DATA_BLOCK "ErrTextList"   // DB371
{ S7_Optimized_Access := 'TRUE' }
// stored: AutoNumber false, MemoryReserve 0
   VAR RETAIN
      language : Array[1..10] of WString[2];   // language for alarm text [ISO639-1]
   END_VAR
   VAR
      writeMessage : Bool;   // write message from program to data block
      err : Array[2000..2205] of Struct   // alarm text
         idProd : UInt;   // producer Id (for Plc: 0=Program_Alarm, 4=SysDiag, 5=MotionControl, 6=Security, 8=GRAPH, 9=ProDiag)
         id : UInt;   // alarm Id
         prio : UInt;   // 0 .. 16 (0-1=info, 2=safety, 3=warning, 4-16=fault)
         alarm : Array[1..8] of WString[150];   // alarm text
      END_STRUCT;
   END_VAR
BEGIN
   language[1] := WSTRING#'de';
   language[2] := WSTRING#'en';
   language[3] := WSTRING#'it';
   language[4] := WSTRING#'fr';
   language[5] := WSTRING#'es';
   err[2031..2040].idProd := 0;
   err[2160..2167].idProd := 0;
   err[2170..2177].idProd := 0;
   err[2180..2187].idProd := 0;
   err[2031..2040].id := 0;
   err[2160..2167].id := 0;
   err[2170..2177].id := 0;
   err[2180..2187].id := 0;
   err[2000..2002].prio := 2;
   err[2004..2005].prio := 2;
   err[2010..2011].prio := 2;
   err[2013..2014].prio := 2;
   err[2016..2017].prio := 2;
   err[2019..2020].prio := 2;
   err[2030..2031].prio := 2;
   err[2032].prio := 0;
   err[2033..2040].prio := 2;
   err[2050].prio := 1;
   err[2052].prio := 0;
   err[2054].prio := 1;
   err[2060].prio := 10;
   err[2075].prio := 2;
   err[2080..2083].prio := 11;
   err[2090..2091].prio := 9;
   err[2100..2102].prio := 10;
   err[2110].prio := 8;
   err[2111].prio := 0;
   err[2120].prio := 12;
   err[2121..2125].prio := 7;
   err[2150].prio := 11;
   err[2151].prio := 10;
   err[2152..2153].prio := 8;
   err[2154].prio := 1;
   err[2156].prio := 1;
   err[2160].prio := 11;
   err[2161].prio := 10;
   err[2162..2163].prio := 8;
   err[2164].prio := 1;
   err[2165].prio := 0;
   err[2166].prio := 1;
   err[2167].prio := 0;
   err[2170].prio := 11;
   err[2171].prio := 10;
   err[2172..2173].prio := 8;
   err[2174].prio := 1;
   err[2175].prio := 0;
   err[2176].prio := 1;
   err[2177].prio := 0;
   err[2180].prio := 11;
   err[2181].prio := 10;
   err[2182..2183].prio := 8;
   err[2184].prio := 1;
   err[2185].prio := 0;
   err[2186].prio := 1;
   err[2187].prio := 0;
   err[2189].prio := 8;
   err[2190].prio := 9;
   err[2000].alarm[1] := WSTRING#'PLC - Not Aus Taster gedrückt am Pc Terminal (-14SB0+HMI.GLD)';
   err[2000].alarm[2] := WSTRING#'PLC - Emergency stop pressed at Pc terminal (-14SB0+HMI.GLD)';
   err[2000].alarm[3] := WSTRING#'PLC - Tasto per arresto di emergenza premuto sul terminale Pc (-14SB0+HMI.GLD)';
   err[2000].alarm[4] := WSTRING#'PLC - Arrêt d`urgence appuyé sur le terminal PC (-14SB0+HMI.GLD)';
   err[2000].alarm[5] := WSTRING#'PLC - Parada de emergencia presionada en terminal Pc (-14SB0+HMI.GLD)';
   err[2001].alarm[1] := WSTRING#'PLC - Not Aus Schlüsselschalter ausgeschalten am Pc Terminal (-14SB1+HMI.GLD)';
   err[2001].alarm[2] := WSTRING#'PLC - Emergency enable key switch off at Pc terminal (-14SB1+HMI.GLD)';
   err[2001].alarm[3] := WSTRING#'PLC - Interruttore a chiave per aresto di emergenza spento sul terminale del PC (-14SB1+HMI.GLD)';
   err[2001].alarm[4] := WSTRING#'PLC - Interrupteur d`urgence désactivé sur le terminal PC (-14SB1+HMI.GLD)';
   err[2001].alarm[5] := WSTRING#'PLC - Interruptor de llave de parada de emergencia apagado en la terminal de la PC (-14SB1+HMI.GLD)';
   err[2002].alarm[1] := WSTRING#'PLC - Quittierung notwendig für Not Aus Taster/Schlüsselschalter am Pc Terminal (-14SB0/1+HMI.GLD)';
   err[2002].alarm[2] := WSTRING#'PLC - Acknowledge required for emergency stop/key switch at Pc terminal (-14SB0/1+HMI.GLD)';
   err[2002].alarm[3] := WSTRING#'PLC - Reset richiesto per pulsante/interrutore di arresto di emergenza sul terminale PC (-14SB0/1+HMI.GLD)';
   err[2002].alarm[4] := WSTRING#'PLC - Reconnaissance nécessaire pour l`arrêt d`urgence/interrupteur à clé sur le terminal PC (-14SB0/1+HMI.GLD)';
   err[2002].alarm[5] := WSTRING#'PLC - Es necesario reiniciar para el botónIinterruptor de emergencia en terminal de PC (-14SB0/1+HMI.GLD)';
   err[2004].alarm[1] := WSTRING#'PLC - Not Aus von externe machine (-XNA+SGV) - aktiv';
   err[2004].alarm[2] := WSTRING#'PLC - Emergency stop from external machine (-XNA+SGV) - active';
   err[2004].alarm[3] := WSTRING#'PLC - Arresto di emergenza da macchina esterna (-XNA+SGV) - attivo';
   err[2004].alarm[4] := WSTRING#'PLC - Arrêt d`urgence depuis une machine externe (-XNA+SGV) - actif';
   err[2004].alarm[5] := WSTRING#'PLC - Parada de emergencia desde máquina externa (-XNA+SGV) - activo';
   err[2005].alarm[1] := WSTRING#'PLC - Not Aus von externe machine (-XNA+SGV) - Quittierung notwendig';
   err[2005].alarm[2] := WSTRING#'PLC - Emergency stop from external machine (-XNA+SGV) - acknowledgement required';
   err[2005].alarm[3] := WSTRING#'PLC - Arresto di emergenza da macchina esterna (-XNA+SGV) - reset necessario';
   err[2005].alarm[4] := WSTRING#'PLC - Arrêt d`urgence depuis une machine externe (-XNA+SGV) - réinitialiser requis';
   err[2005].alarm[5] := WSTRING#'PLC - Parada de emergencia desde máquina externa (-XNA+SGV) - es necesario reiniciar';
   err[2010].alarm[1] := WSTRING#'PLC - Sicherheitsschalter -14SS1.TL+SGV bei Scanner für visuelle Beurteilung oben links - open';
   err[2010].alarm[2] := WSTRING#'PLC - Safety switch -14SS1.TL+SGV at scanner for visual measurement top left - open';
   err[2010].alarm[3] := WSTRING#'PLC - Interruttore di sicurezza -14SS1.TL+SGV sullo scanner per misurazione visiva in alto a sinistra - aperto';
   err[2010].alarm[4] := WSTRING#'PLC - interrupteur de sécurité -14SS1.TL+SGV au scanner pour mesure visuelle en haut à gauche - ouvert';
   err[2010].alarm[5] := WSTRING#'PLC - interruptor de seguridad -14SS1.TL+SGV en el escáner para medición visual arriba a la izquierda - abierto';
   err[2011].alarm[1] := WSTRING#'PLC - Sicherheitsschalter -14SS1.TL+SGV bei Scanner für visuelle Beurteilung oben links - Quittierung notwendig';
   err[2011].alarm[2] := WSTRING#'PLC - safety switch -14SS1.TL+SGV at scanner for visual measurement top left - acknowledge required';
   err[2011].alarm[3] := WSTRING#'PLC - Interruttore di sicurezza -14SS1.TL+SGV sullo scanner per misurazione visiva in alto a sinistra - reset necessario';
   err[2011].alarm[4] := WSTRING#'PLC - interrupteur de sécurité -14SS1.TL+SGV au scanner pour mesure visuelle en haut à gauche - réinitialiser requis';
   err[2011].alarm[5] := WSTRING#'PLC - interruptor de seguridad -14SS1.TL+SGV en el escáner para medición visual arriba a la izquierda - es necesario reiniciar';
   err[2013].alarm[1] := WSTRING#'PLC - Sicherheitsschalter -14SS1.BL+SGV bei Scanner für visuelle Beurteilung unten links - open';
   err[2013].alarm[2] := WSTRING#'PLC - Safety switch -14SS1.BL+SGV at scanner for visual measurement bottom left - open';
   err[2013].alarm[3] := WSTRING#'PLC - Interruttore di sicurezza -14SS1.BL+SGV sullo scanner per misurazione visiva in basso a sinistra - aperto';
   err[2013].alarm[4] := WSTRING#'PLC - interrupteur de sécurité -14SS1.BL+SGV au scanner pour mesure visuelle en bas à gauche - ouvert';
   err[2013].alarm[5] := WSTRING#'PLC - interruptor de seguridad -14SS1.BL+SGV en el escáner para medición visual abajoa la izquierda - abierto';
   err[2014].alarm[1] := WSTRING#'PLC - Sicherheitsschalter -14SS1.BL+SGV bei Scanner für visuelle Beurteilung unten links - Quittierung notwendig';
   err[2014].alarm[2] := WSTRING#'PLC - Safety switch -14SS1.BL+SGV at scanner for visual measurement bottom left - acknowledge required';
   err[2014].alarm[3] := WSTRING#'PLC - Interruttore di sicurezza -14SS1.BL+SGV sullo scanner per misurazione visiva in basso a sinistra - reset necessario';
   err[2014].alarm[4] := WSTRING#'PLC - interrupteur de sécurité -14SS1.BL+SGV au scanner pour mesure visuelle en bas à gauche - réinitialiser requis';
   err[2014].alarm[5] := WSTRING#'PLC - interruptor de seguridad -14SS1.BL+SGV en el escáner para medición visual abajoa la izquierda - es necesario reiniciar';
   err[2016].alarm[1] := WSTRING#'PLC - Sicherheitsschalter -14SS1.TR+SGV bei Scanner für visuelle Beurteilung oben rechts- open';
   err[2016].alarm[2] := WSTRING#'PLC - Safety switch -14SS1.TR+SGV at scanner for visual measurement top right - open';
   err[2016].alarm[3] := WSTRING#'PLC - Interruttore di sicurezza -14SS1.TR+SGV sullo scanner per misurazione visiva in alto a destra - aperto';
   err[2016].alarm[4] := WSTRING#'PLC - interrupteur de sécurité -14SS1.TR+SGV au scanner pour mesure visuelle en haut à droite - ouvert';
   err[2016].alarm[5] := WSTRING#'PLC - interruptor de seguridad -14SS1.TR+SGV en el escáner para medición visual arriba a la derecha - abierto';
   err[2017].alarm[1] := WSTRING#'PLC - Sicherheitsschalter -14SS1.TR+SGV bei Scanner für visuelle Beurteilung oben rechts- Quittierung notwendig';
   err[2017].alarm[2] := WSTRING#'PLC - Safety switch -14SS1.TR+SGV at scanner for visual measurement top right -  acknowledge required';
   err[2017].alarm[3] := WSTRING#'PLC - Interruttore di sicurezza -14SS1.TR+SGV sullo scanner per misurazione visiva in alto a destra - reset necessario';
   err[2017].alarm[4] := WSTRING#'PLC - interrupteur de sécurité -14SS1.TR+SGV au scanner pour mesure visuelle en haut à droite - réinitialiser requis';
   err[2017].alarm[5] := WSTRING#'PLC - interruptor de seguridad -14SS1.TR+SGV en el escáner para medición visual arriba a la derecha - es necesario reiniciar';
   err[2019].alarm[1] := WSTRING#'PLC - Sicherheitsschalter -14SS1.BR+SGV bei Scanner für visuelle Beurteilung unten rechts - open';
   err[2019].alarm[2] := WSTRING#'PLC - Safety switch -14SS1.BR+SGV at scanner for visual measurement bottom right - open';
   err[2019].alarm[3] := WSTRING#'PLC - Interruttore di sicurezza -14SS1.BR+SGV sullo scanner per misurazione visiva in basso a destra - aperto';
   err[2019].alarm[4] := WSTRING#'PLC - interrupteur de sécurité -14SS1.BR+SGV au scanner pour mesure visuelle en bas à droite - ouvert';
   err[2019].alarm[5] := WSTRING#'PLC - interruptor de seguridad -14SS1.BR+SGV en el escáner para medición visual abajo a la derecha - abierto';
   err[2020].alarm[1] := WSTRING#'PLC - Sicherheitsschalter -14SS1.BR+SGV bei Scanner für visuelle Beurteilung unten rechts - Quittierung notwendig';
   err[2020].alarm[2] := WSTRING#'PLC - Safety switch -14SS1.BR+SGV at scanner for visual measurement bottom right -  acknowledge required';
   err[2020].alarm[3] := WSTRING#'PLC - Interruttore di sicurezza -14SS1.BR+SGV sullo scanner per misurazione visiva in basso a destra - reset necessario';
   err[2020].alarm[4] := WSTRING#'PLC - interrupteur de sécurité -14SS1.BR+SGV au scanner pour mesure visuelle en bas à droite - réinitialiser requis';
   err[2020].alarm[5] := WSTRING#'PLC - interruptor de seguridad -14SS1.BR+SGV en el escáner para medición visual abajo a la derecha - es necesario reiniciar';
   err[2030].alarm[1] := WSTRING#'PLC - Sicherheitsschalter -14SS1.TL+SGX bei Scanner für X-Ray oben links - open';
   err[2030].alarm[2] := WSTRING#'PLC - Safety switch -14SS1.TL+SGX at scanner for X-Ray top left - open';
   err[2030].alarm[3] := WSTRING#'PLC - Interruttore di sicurezza -14SS1.TL+SGX sullo scanner per X-Ray in alto a sinistra - aperto';
   err[2030].alarm[4] := WSTRING#'PLC - interrupteur de sécurité -14SS1.TL+SGX au scanner pour X-Ray en haut à gauche - ouvert';
   err[2030].alarm[5] := WSTRING#'PLC - interruptor de seguridad -14SS1.TL+SGX en el escáner para X-Ray arriba a la izquierda - abierto';
   err[2030].alarm[6..8] := WSTRING#'';
   err[2031].alarm[1] := WSTRING#'PLC - Sicherheitsschalter -14SS1.TL+SGX bei Scanner für X-Ray oben links - Quittierung notwendig';
   err[2031].alarm[2] := WSTRING#'PLC - safety switch -14SS1.TL+SGX at scanner for X-Ray top left - acknowledge required';
   err[2031].alarm[3] := WSTRING#'PLC - Interruttore di sicurezza -14SS1.TL+SGX sullo scanner per X-Ray in alto a sinistra - reset necessario';
   err[2031].alarm[4] := WSTRING#'PLC - interrupteur de sécurité -14SS1.TL+SGX au scanner pour X-Ray en haut à gauche - réinitialiser requis';
   err[2031].alarm[5] := WSTRING#'PLC - interruptor de seguridad -14SS1.TL+SGX en el escáner para X-Ray arriba a la izquierda - es necesario reiniciar';
   err[2031].alarm[6..8] := WSTRING#'';
   err[2032].alarm[1..8] := WSTRING#'';
   err[2033].alarm[1] := WSTRING#'PLC - Sicherheitsschalter -14SS1.BL+SGX bei Scanner für X-Ray unten links - open';
   err[2033].alarm[2] := WSTRING#'PLC - Safety switch -14SS1.BL+SGX at scanner for X-Ray bottom left - open';
   err[2033].alarm[3] := WSTRING#'PLC - Interruttore di sicurezza -14SS1.BL+SGX sullo scanner per X-Ray in basso a sinistra - aperto';
   err[2033].alarm[4] := WSTRING#'PLC - interrupteur de sécurité -14SS1.BL+SGX au scanner pour X-Ray en bas à gauche - ouvert';
   err[2033].alarm[5] := WSTRING#'PLC - interruptor de seguridad -14SS1.BL+SGX en el escáner para X-Ray abajoa la izquierda - abierto';
   err[2033].alarm[6..8] := WSTRING#'';
   err[2034].alarm[1] := WSTRING#'PLC - Sicherheitsschalter -14SS1.BL+SGX bei Scanner für X-Ray unten links - Quittierung notwendig';
   err[2034].alarm[2] := WSTRING#'PLC - Safety switch -14SS1.BL+SGX at scanner for X-Rayt bottom left - acknowledge required';
   err[2034].alarm[3] := WSTRING#'PLC - Interruttore di sicurezza -14SS1.BL+SGX sullo scanner per X-Ray in basso a sinistra - reset necessario';
   err[2034].alarm[4] := WSTRING#'PLC - interrupteur de sécurité -14SS1.BL+SGX au scanner pour X-Ray en bas à gauche - réinitialiser requis';
   err[2034].alarm[5] := WSTRING#'PLC - interruptor de seguridad -14SS1.BL+SGX en el escáner para X-Ray abajoa la izquierda - es necesario reiniciar';
   err[2034].alarm[6..8] := WSTRING#'';
   err[2035].alarm[1..8] := WSTRING#'';
   err[2036].alarm[1] := WSTRING#'PLC - Sicherheitsschalter -14SS1.TR+SGX bei Scanner für X-Ray oben rechts- open';
   err[2036].alarm[2] := WSTRING#'PLC - Safety switch -14SS1.TR+SGX at scanner for X-Ray top right - open';
   err[2036].alarm[3] := WSTRING#'PLC - Interruttore di sicurezza -14SS1.TR+SGX sullo scanner per X-Ray in alto a destra - aperto';
   err[2036].alarm[4] := WSTRING#'PLC - interrupteur de sécurité -14SS1.TR+SGX au scanner pour X-Ray en haut à droite - ouvert';
   err[2036].alarm[5] := WSTRING#'PLC - interruptor de seguridad -14SS1.TR+SGX en el escáner para X-Ray arriba a la derecha - abierto';
   err[2036].alarm[6..8] := WSTRING#'';
   err[2037].alarm[1] := WSTRING#'PLC - Sicherheitsschalter -14SS1.TR+SGX bei Scanner für X-Ray oben rechts- Quittierung notwendig';
   err[2037].alarm[2] := WSTRING#'PLC - Safety switch -14SS1.TR+SGX at scanner for X-Ray top right -  acknowledge required';
   err[2037].alarm[3] := WSTRING#'PLC - Interruttore di sicurezza -14SS1.TR+SGX sullo scanner per X-Ray in alto a destra - reset necessario';
   err[2037].alarm[4] := WSTRING#'PLC - interrupteur de sécurité -14SS1.TR+SGX au scanner pour X-Ray en haut à droite - réinitialiser requis';
   err[2037].alarm[5] := WSTRING#'PLC - interruptor de seguridad -14SS1.TR+SGX en el escáner para X-Ray arriba a la derecha - es necesario reiniciar';
   err[2037].alarm[6..8] := WSTRING#'';
   err[2038].alarm[1..8] := WSTRING#'';
   err[2039].alarm[1] := WSTRING#'PLC - Sicherheitsschalter -14SS1.BR+SGX bei Scanner für X-Ray unten rechts - open';
   err[2039].alarm[2] := WSTRING#'PLC - Safety switch -14SS1.BR+SGX at scanner for X-Ray bottom right - open';
   err[2039].alarm[3] := WSTRING#'PLC - Interruttore di sicurezza -14SS1.BR+SGX sullo scanner per X-Ray in basso a destra - aperto';
   err[2039].alarm[4] := WSTRING#'PLC - interrupteur de sécurité -14SS1.BR+SGX au scanner pour X-Ray en bas à droite - ouvert';
   err[2039].alarm[5] := WSTRING#'PLC - interruptor de seguridad -14SS1.BR+SGX en el escáner para X-Ray abajo a la derecha - abierto';
   err[2039].alarm[6..8] := WSTRING#'';
   err[2040].alarm[1] := WSTRING#'PLC - Sicherheitsschalter -14SS1.BR+SGX bei Scanner für X-Ray unten rechts - Quittierung notwendig';
   err[2040].alarm[2] := WSTRING#'PLC - Safety switch -14SS1.BR+SGX at scanner for X-Ray bottom right -  acknowledge required';
   err[2040].alarm[3] := WSTRING#'PLC - Interruttore di sicurezza -14SS1.BR+SGX sullo scanner per X-Ray in basso a destra - reset necessario';
   err[2040].alarm[4] := WSTRING#'PLC - interrupteur de sécurité -14SS1.BR+SGX au scanner pour X-Ray en bas à droite - réinitialiser requis';
   err[2040].alarm[5] := WSTRING#'PLC - interruptor de seguridad -14SS1.BR+SGX en el escáner para X-Ray abajo a la derecha - es necesario reiniciar';
   err[2050].alarm[1] := WSTRING#'PLC - Schlüsselschalter für Einrichtbetrieb am Scanner links aktiviert (-14SB1+SSTL)';
   err[2050].alarm[2] := WSTRING#'PLC - setting mode key switch at scanner left active (-14SB1+SSTL)';
   err[2050].alarm[3] := WSTRING#'PLC - Interruttore a chiave per la modalità di impostazione attivato sullo scanner a sinistra (-14SB1+SSTL)';
   err[2050].alarm[4] := WSTRING#'PLC - commutateur à clé du mode de réglage à gauche du scanner actif (-14SB1+SSTL)';
   err[2050].alarm[5] := WSTRING#'PLC - interruptor de modo de ajuste a la izquierda del escáner activo (-14SB1+SSTL)';
   err[2052].alarm[1] := WSTRING#'PLC - Taster für Freigabe Verstellungen am Scanner links aktiviert (-14SB2+SSTL)';
   err[2052].alarm[2] := WSTRING#'PLC - button to enable adjustments at scanner left active (-14SB21+SSTL)';
   err[2052].alarm[3] := WSTRING#'PLC - pulsante per abilitare le assi attivato sullo scanner a sinistra (-14SB2+SSTL)';
   err[2052].alarm[4] := WSTRING#'PLC - bouton pour activer les réglages à gauche du scanner actif (-14SB2+SSTL)';
   err[2052].alarm[5] := WSTRING#'PLC - botón para habilitar ajustes a la izquierda del escáner activo (-14SB2+SSTL)';
   err[2054].alarm[1] := WSTRING#'PLC - Kühlgeräte wurden am Scanner rechts deaktiviert (-14SB2+SSTL)';
   err[2054].alarm[2] := WSTRING#'PLC - air-conditioning is switched off at scanner right (-0SH1+SSTR)';
   err[2054].alarm[3] := WSTRING#'PLC - l`aria condizionata è stata spenta sullo scanner a destra (-14SB2+SSTL)';
   err[2054].alarm[4] := WSTRING#'PLC - la climatisation est éteinte au niveau du scanner à droite (-14SB2+SSTL)';
   err[2054].alarm[5] := WSTRING#'PLC - El aire acondicionado está apagado en el escáner a la derecha (-14SB2+SSTL)';
   err[2060].alarm[1] := WSTRING#'PLC - Störung Sicherheitsmodule';
   err[2060].alarm[2] := WSTRING#'PLC - fault safety modules plc';
   err[2060].alarm[3] := WSTRING#'PLC - errore sui moduli di sicurezza';
   err[2060].alarm[4] := WSTRING#'PLC - modules de sécurité contre les défauts';
   err[2060].alarm[5] := WSTRING#'PLC - módulos de seguridad contra fallas';
   err[2075].alarm[1] := WSTRING#'PLC - Sicherheitsbereich Extern oder Intern ausgeschalten - Quittierung notwendig';
   err[2075].alarm[2] := WSTRING#'PLC - safety area internal/external switched off - acknowledge required';
   err[2075].alarm[3] := WSTRING#'PLC - area di sicurezza interna/esterna spenta- reset necessario';
   err[2075].alarm[4] := WSTRING#'PLC - zone de sécurité interne/externe désactivée - réinitialiser requis';
   err[2075].alarm[5] := WSTRING#'PLC - area de seguridad interna/externa apagada - es necesario reiniciar';
   err[2080].alarm[1] := WSTRING#'PLC - Störung Rückführung Sicherheitsbereich - Bereich laser (-14KA1+SGV)';
   err[2080].alarm[2] := WSTRING#'PLC - fault safety feedback monitoring - area laser (-14KA1+SGV)';
   err[2080].alarm[3] := WSTRING#'PLC - errore monitoraggio feedback di sicurezza - area laser (-14KA1+SGV)';
   err[2080].alarm[4] := WSTRING#'PLC - défaut surveillance de la sécurité - zone laser (-14KA1+SGV)';
   err[2080].alarm[5] := WSTRING#'PLC - fallo de monitoreo de retroalimentación de seguridad - área de láser (-14KA1+SGV)';
   err[2081].alarm[1] := WSTRING#'PLC - Störung Rückführung Sicherheitsbereich - Bereich Verstellung (-14KA2+SGV)';
   err[2081].alarm[2] := WSTRING#'PLC - fault safety feedback monitoring - area adjustment (-14KA2+SGV)';
   err[2081].alarm[3] := WSTRING#'PLC - errore monitoraggio feedback di sicurezza - area posizionamento (-14KA2+SGV)';
   err[2081].alarm[4] := WSTRING#'PLC - défaut surveillance de la sécurité - zone réglage (-14KA2+SGV)';
   err[2081].alarm[5] := WSTRING#'PLC - fallo de monitoreo de retroalimentación de seguridad - área de ajuste (-14KA2+SGV)';
   err[2082].alarm[1] := WSTRING#'PLC - Störung Rückführung Sicherheitsbereich - Bereich Verstellung LINMOT (8U1+SGV)';
   err[2082].alarm[2] := WSTRING#'PLC - fault safety feedback monitoring - area adjustment LINMOT (8U1+SGV)';
   err[2082].alarm[3] := WSTRING#'PLC - errore monitoraggio feedback di sicurezza - area posizionamento LINMOT (8U1+SGV)';
   err[2082].alarm[4] := WSTRING#'PLC - défaut surveillance de la sécurité - zone réglage LINMOT (8U1+SGV)';
   err[2082].alarm[5] := WSTRING#'PLC - fallo de monitoreo de retroalimentación de seguridad - área de ajuste LINMOT (8U1+SGV)';
   err[2083].alarm[1] := WSTRING#'PLC - Störung Rückführung Sicherheitsbereich - Bereich X-Ray (-5AX1+SGX)';
   err[2083].alarm[2] := WSTRING#'PLC - fault safety feedback monitoring - area X-Ray (-5AX1+SGX)';
   err[2083].alarm[3] := WSTRING#'PLC - errore monitoraggio feedback di sicurezza - area X-Ray (-5AX1+SGX)';
   err[2083].alarm[4] := WSTRING#'PLC - défaut surveillance de la sécurité - zone X-Ray (-5AX1+SGX)';
   err[2083].alarm[5] := WSTRING#'PLC - fallo de monitoreo de retroalimentación de seguridad - área X-Ray (-5AX1+SGX)';
   err[2090].alarm[1] := WSTRING#'PLC - Störung Lichtschranke im Scanner für visuelle Beurteilung (-1BTR2+SGV)';
   err[2090].alarm[2] := WSTRING#'PLC - fault light barrier in scanner for visual measurement (-1BTR2+SGV)';
   err[2090].alarm[3] := WSTRING#'PLC - errore sensore nel scanner per misurazione visiva (-1BTR2+SGV)';
   err[2090].alarm[4] := WSTRING#'PLC - défaut capteur dans le scanner pour la mesure visuelle (-1BTR2+SGV)';
   err[2090].alarm[5] := WSTRING#'PLC - fallo de sensor en escáner para medición visual (-1BTR2+SGV)';
   err[2091].alarm[1] := WSTRING#'PLC - Störung Lichtschranke vor Scanner für X-Ray (-1BTR2+SGX)';
   err[2091].alarm[2] := WSTRING#'PLC - fault light barrier before scanner for X-Ray (-1BTR2+SGX)';
   err[2091].alarm[3] := WSTRING#'PLC - errore sensore prime dello scanner per X-Ray (-1BTR2+SGX)';
   err[2091].alarm[4] := WSTRING#'PLC - défaut capteur avant le scanner pour X-Ray (-1BTR2+SGX)';
   err[2091].alarm[5] := WSTRING#'PLC - fallo de sensor antes escáner para X-Ray (-1BTR2+SGX)';
   err[2100].alarm[1] := WSTRING#'PLC - Störung Encoder vor Scanner (-1BCI1+GLD)';
   err[2100].alarm[2] := WSTRING#'PLC - fault encoder before scanner (-1BCI1+GLD)';
   err[2100].alarm[3] := WSTRING#'PLC - errore encoder davanti allo scanner (-1BCI1+GLD)';
   err[2100].alarm[4] := WSTRING#'PLC - défaut codeur avant le scanner (-1BCI1+GLD)';
   err[2100].alarm[5] := WSTRING#'PLC - fallo de codificador antes escáner (-1BCI1+GLD)';
   err[2101].alarm[1] := WSTRING#'PLC - Störung Encoder im Scanner (-1BCM1+GLD)';
   err[2101].alarm[2] := WSTRING#'PLC - fault encoder in scanner (-1BCM1+GLD)';
   err[2101].alarm[3] := WSTRING#'PLC - errore encoder nello scanner (-1BCM1+GLD)';
   err[2101].alarm[4] := WSTRING#'PLC - défaut codeur dans le scanner (-1BCM1+GLD)';
   err[2101].alarm[5] := WSTRING#'PLC - fallo de codificador en escáner (-1BCM1+GLD)';
   err[2102].alarm[1] := WSTRING#'PLC - Störung Encoder nach Scanner (-1BCO1+GLD)';
   err[2102].alarm[2] := WSTRING#'PLC - fault encoder after scanner (-1BCO1+GLD)';
   err[2102].alarm[3] := WSTRING#'PLC - errore encoder dopo lo scanner (-1BCO1+GLD)';
   err[2102].alarm[4] := WSTRING#'PLC - défaut codeur après le scanner (-1BCO1+GLD)';
   err[2102].alarm[5] := WSTRING#'PLC - fallo de codificador después del escáner (-1BCO1+GLD)';
   err[2110].alarm[1] := WSTRING#'PLC - Störung Kommunikation mit Goldeneye Pc';
   err[2110].alarm[2] := WSTRING#'PLC - fault communication with Goldeneye Pc';
   err[2110].alarm[3] := WSTRING#'PLC - errore comunicazione con Goldeneye Pc';
   err[2110].alarm[4] := WSTRING#'PLC - défaut communication avec Goldeneye Pc';
   err[2110].alarm[5] := WSTRING#'PLC - fallo comunicación con Goldeneye Pc';
   err[2111].alarm[1] := WSTRING#'PLC - Keine Freigabe vom Goldeneye Pc für den Einzug';
   err[2111].alarm[2] := WSTRING#'PLC - no release from Goldeneye Pc to infeed';
   err[2111].alarm[3] := WSTRING#'PLC - nessun permesso dal Goldeneye Pc per alimentazione ';
   err[2111].alarm[4] := WSTRING#'PLC - pas de sortie de Goldeneye PC pour infeed';
   err[2111].alarm[5] := WSTRING#'PLC - no hay liberación de Goldeneye Pc para la entrada';
   err[2120].alarm[1] := WSTRING#'PLC - Störung elektronischer Schutzschalter (-0F1.1+SGV)';
   err[2120].alarm[2] := WSTRING#'PLC - fault electronic circuit breaker (-0F1.1+SGV)';
   err[2120].alarm[3] := WSTRING#'PLC - errore interruttore elettronico (-0F1.1+SGV)';
   err[2120].alarm[4] := WSTRING#'PLC - défaut disjoncteur électronique (-0F1.1+SGV)';
   err[2120].alarm[5] := WSTRING#'PLC - fallo disyuntor electrónico (-0F1.1+SGV)';
   err[2121].alarm[1] := WSTRING#'PLC - Störung Kühlgerät 1 bei Scanner für visuelle Beurteilung (-0E1+SGV)';
   err[2121].alarm[2] := WSTRING#'PLC - fault air-conditioning unit 1 for scannerhousing visual measurement (-0E1+SGV)';
   err[2121].alarm[3] := WSTRING#'PLC - errore unità di raffreddamento 1 per scanner per misurazione visiva (-0E1+SGV)';
   err[2121].alarm[4] := WSTRING#'PLC - défaut unité de refroidissement 1 chez scanner pour mesure visuelle (-0E1+SGV)';
   err[2121].alarm[5] := WSTRING#'PLC - fallo unidad de refrigeración 1 para escáner para medición visual (-0E1+SGV)';
   err[2122].alarm[1] := WSTRING#'PLC - Störung Kühlgerät bei Scanner für X-Ray (-0E2+SGX)';
   err[2122].alarm[2] := WSTRING#'PLC - fault air-conditioning unit for scannerhousing  X-Ray (-0E2+SGX)';
   err[2122].alarm[3] := WSTRING#'PLC - errore unità di raffreddamento per scanner per X-Ray (-0E2+SGX)';
   err[2122].alarm[4] := WSTRING#'PLC - défaut unité de refroidissement chez scanner pour X-Ray (-0E2+SGX)';
   err[2122].alarm[5] := WSTRING#'PLC - fallo unidad de refrigeración para escáner para X-Ray (-0E2+SGX)';
   err[2123].alarm[1] := WSTRING#'PLC - Störung Kühlgerät 2 bei Scanner für visuelle Beurteilung (-0E1.1+SGV)';
   err[2123].alarm[2] := WSTRING#'PLC - fault air-conditioning unit 2 for scannerhousing visual measurement (-0E1.1+SGV)';
   err[2123].alarm[3] := WSTRING#'PLC - errore unità di raffreddamento 2 per scanner per misurazione visiva (-0E1.1+SGV)';
   err[2123].alarm[4] := WSTRING#'PLC - défaut unité de refroidissement 2 chez scanner pour mesure visuelle (-0E1.1+SGV)';
   err[2123].alarm[5] := WSTRING#'PLC - fallo unidad de refrigeración 2 para escáner para medición visual (-0E1.1+SGV)';
   err[2124].alarm[1] := WSTRING#'PLC - Störung Entfeuchter bei Scanner für (-0E1.2+SGV)';
   err[2124].alarm[2] := WSTRING#'PLC - fault dehumidifier for scannerhousing (-0E1.2+SGV)';
   err[2124].alarm[3] := WSTRING#'PLC - errore deumidificatore per scanner (-0E1.2+SGV)';
   err[2124].alarm[4] := WSTRING#'PLC - défaut déshumidificateur chez scanner (-0E1.2+SGV)';
   err[2124].alarm[5] := WSTRING#'PLC - fallo deshumidificador para escáner (-0E1.2+SGV)';
   err[2125].alarm[1] := WSTRING#'PLC - Störung Kommunikationsschnittstelle zwischen Pc und Sps ist unterschiedlich';
   err[2125].alarm[2] := WSTRING#'PLC - fault communication interface between Pc and Plc is different';
   err[2125].alarm[3] := WSTRING#'PLC - errore l`interfaccia di comunicazione tra Pc e Plc è diversa';
   err[2125].alarm[4] := WSTRING#'PLC - défaut l`interface de communication entre le PC et Plc est différente';
   err[2125].alarm[5] := WSTRING#'PLC - fallo La interfaz de comunicación entre PC y PLC es diferente';
   err[2140].alarm[1] := WSTRING#'PLC - Verstellung Scanner wurde temporär deaktiviert, kann nur mehr manuel verfahren werden (-8M1.B+SGV)';
   err[2140].alarm[2] := WSTRING#'PLC - adjustment scannerhousing is deactivated temporaly, you can move only manualy (-8M1.B+SGV)';
   err[2140].alarm[3] := WSTRING#'PLC - posizionamento scanner è temporaneamente disattivato, è possibile muoverlo solo manualmente (-8M1.B+SGV)';
   err[2140].alarm[4] := WSTRING#'PLC - positionnement de scanner est temporairement désactivé, vous ne pouvez le déplacer que manuellement (-8M1.B+SGV)';
   err[2140].alarm[5] := WSTRING#'PLC - el ajuste de del escáner se desactiva temporalmente, solo se puede mover manualmente (-8M1.B+SGV)';
   err[2141].alarm[1] := WSTRING#'PLC - Verstellung Messbalken oben wurde temporär deaktiviert, kann nur mehr manuel verfahren werden (-8M1.T+SGV)';
   err[2141].alarm[2] := WSTRING#'PLC - adjustment metering bar top is deactivated temporaly, you can move only manualy (-8M1.T+SGV)';
   err[2141].alarm[3] := WSTRING#'PLC - posizionamento barra di misura superiore è temporaneamente disattivato, è possibile muoverlo solo manualmente (-8M1.T+SGV)';
   err[2141].alarm[4] := WSTRING#'PLC - positionnement de barre de mesure supérieure est temporairement désactivé, vous ne pouvez le déplacer que manuellement (-8M1.T+SGV)';
   err[2141].alarm[5] := WSTRING#'PLC - el ajuste de barra de medición superior se desactiva temporalmente, solo se puede mover manualmente (-8M1.T+SGV)';
   err[2142].alarm[1] := WSTRING#'PLC - Verstellung Messbalken links wurde temporär deaktiviert, kann nur mehr manuel verfahren werden (-8M1.L+SGV)';
   err[2142].alarm[2] := WSTRING#'PLC - adjustment metering bar left is deactivated temporaly, you can move only manualy (-8M1.L+SGV)';
   err[2142].alarm[3] := WSTRING#'PLC - posizionamento barra di misura di sinistra è temporaneamente disattivato, è possibile muoverlo solo manualmente (-8M1.L+SGV)';
   err[2142].alarm[4] := WSTRING#'PLC - positionnement de barre de mesure gauche est temporairement désactivé, vous ne pouvez le déplacer que manuellement (-8M1L+SGV)';
   err[2142].alarm[5] := WSTRING#'PLC - el ajuste de barra de medición izquierda se desactiva temporalmente, solo se puede mover manualmente (-8M1.L+SGV)';
   err[2143].alarm[1] := WSTRING#'PLC - Verstellung Messbalken rechts wurde temporär deaktiviert, kann nur mehr manuel verfahren werden (-8M1.R+SGV)';
   err[2143].alarm[2] := WSTRING#'PLC - adjustment metering bar right is deactivated temporaly, you can move only manualy (-8M1.R+SGV)';
   err[2143].alarm[3] := WSTRING#'PLC - posizionamento barra di misura di destra è temporaneamente disattivato, è possibile muoverlo solo manualmente (-8M1.R+SGV)';
   err[2143].alarm[4] := WSTRING#'PLC - positionnement de barre de mesure à droite est temporairement désactivé, vous ne pouvez le déplacer que manuellement (-8M1.R+SGV)';
   err[2143].alarm[5] := WSTRING#'PLC - el ajuste de barra de medición derecha se desactiva temporalmente, solo se puede mover manualmente (-8M1.R+SGV)';
   err[2144].alarm[1] := WSTRING#'PLC - Kühlgerät 1 bei Scanner für visuelle Beurteilung wurde temporär deaktiviert (-0E1+SGV)';
   err[2144].alarm[2] := WSTRING#'PLC - air-conditioning unit 1 for scannerhousing visual measurement is deactivated temporaly (-0E1+SGV)';
   err[2144].alarm[3] := WSTRING#'PLC - unità di raffreddamento 1 per scanner per misurazione visiva è temporaneamente disattivato (-0E1+SGV)';
   err[2144].alarm[4] := WSTRING#'PLC - unité de refroidissement 1 chez scanner pour mesure visuelle est temporairement désactivé (-0E1+SGV)';
   err[2144].alarm[5] := WSTRING#'PLC - unidad de refrigeración 1 para escáner para medición visual se desactiva temporalmente (-0E1+SGV)';
   err[2145].alarm[1] := WSTRING#'PLC - Kühlgerät 2 bei Scanner für visuelle Beurteilung wurde temporär deaktiviert (-0E1.1+SGV)';
   err[2145].alarm[2] := WSTRING#'PLC - air-conditioning unit 2 for scannerhousing visual measurement is deactivated temporaly (-0E1.1+SGV)';
   err[2145].alarm[3] := WSTRING#'PLC - unità di raffreddamento 2 per scanner per misurazione visiva è temporaneamente disattivato (-0E1.1+SGV)';
   err[2145].alarm[4] := WSTRING#'PLC - unité de refroidissement 2 chez scanner pour mesure visuelle est temporairement désactivé (-0E1.1+SGV)';
   err[2145].alarm[5] := WSTRING#'PLC - unidad de refrigeración 2 para escáner para medición visual se desactiva temporalmente (-0E1.1+SGV)';
   err[2146].alarm[1] := WSTRING#'PLC - Kühlgerät bei Scanner für X-Ray wurde temporär deaktiviert (-0E2+SGX)';
   err[2146].alarm[2] := WSTRING#'PLC - air-conditioning unit for scannerhousing X-Ray measurement is deactivated temporaly (-0E2+SGX)';
   err[2146].alarm[3] := WSTRING#'PLC - unità di raffreddamento per scanner per X-Ray è temporaneamente disattivato (-0E2+SGX)';
   err[2146].alarm[4] := WSTRING#'PLC - unité de refroidissement chez scanner pour X-Ray est temporairement désactivé (-0E2+SGX)';
   err[2146].alarm[5] := WSTRING#'PLC - unidad de refrigeración 1 para escáner paraX-Ray se desactiva temporalmente (-0E2+SGX)';
   err[2147].alarm[1] := WSTRING#'PLC - Entfeuchter bei Scanner wurde temporär deaktiviert (-0E3+SGX)';
   err[2147].alarm[2] := WSTRING#'PLC - dehumidifier for scannerhousing is deactivated temporaly (-0E3+SGX)';
   err[2147].alarm[3] := WSTRING#'PLC - deumidificatore per scanner è temporaneamente disattivato (-0E3+SGX)';
   err[2147].alarm[4] := WSTRING#'PLC - déshumidificateur chez scanner est temporairement désactivé (-0E3+SGX)';
   err[2147].alarm[5] := WSTRING#'PLC - deshumidificador para escáner se desactiva temporalmente (-0E3+SGX)';
   err[2150].alarm[1] := WSTRING#'PLC - Störung Verstellung Scanner (-8M1.B+SGV)';
   err[2150].alarm[2] := WSTRING#'PLC - fault adjustment scannerhousing (-8M1.B+SGV)';
   err[2150].alarm[3] := WSTRING#'PLC - errore posizionamento scanner (-8M1.B+SGV)';
   err[2150].alarm[4] := WSTRING#'PLC - défaut positionnement de scanner (-8M1.B+SGV)';
   err[2150].alarm[5] := WSTRING#'PLC - fallo el ajuste de del escáner (-8M1.B+SGV)';
   err[2151].alarm[1] := WSTRING#'PLC - Störung Encoder - Verstellung Scanner (-8B1.B+SGV)';
   err[2151].alarm[2] := WSTRING#'PLC - fault encoder - adjustment scannerhousing (-8B1.B+SGV)';
   err[2151].alarm[3] := WSTRING#'PLC - errore encoder - posizionamento scanner (-8B1.B+SGV)';
   err[2151].alarm[4] := WSTRING#'PLC - défaut codeur - positionnement de scanner (-8B1.B+SGV)';
   err[2151].alarm[5] := WSTRING#'PLC - fallo codificador - el ajuste de del escáner (-8B1.B+SGV)';
   err[2152].alarm[1] := WSTRING#'PLC - Störung Sensor Endstellung links - Verstellung Scanner (-8S1.B+SGV)';
   err[2152].alarm[2] := WSTRING#'PLC - fault sensor limit switch position left - adjustment scannerhousing (-8S1.B+SGV)';
   err[2152].alarm[3] := WSTRING#'PLC - errore sensore posizione sinistra - posizionamento scanner (-8S1.B+SGV)';
   err[2152].alarm[4] := WSTRING#'PLC - défaut capteur position du fin de course à gauche - positionnement de scanner (-8S1.B+SGV)';
   err[2152].alarm[5] := WSTRING#'PLC - fallo sensor posición de límite a la izquierda - el ajuste de del escáner (-8S1.B+SGV)';
   err[2153].alarm[1] := WSTRING#'PLC - Störung Sensor Endstellung rechts - Verstellung Scanner (-8S2.B+SGV)';
   err[2153].alarm[2] := WSTRING#'PLC - fault sensor limit switch position right - adjustment scannerhousing (-8S2.B+SGV)';
   err[2153].alarm[3] := WSTRING#'PLC - errore sensore posizione destra - posizionamento scanner (-8S2.B+SGV)';
   err[2153].alarm[4] := WSTRING#'PLC - défaut capteur position du fin de course à droite - positionnement de scanner (-8S2.B+SGV)';
   err[2153].alarm[5] := WSTRING#'PLC - fallo sensor posición de límite a la derecha - el ajuste de del escáner (-8S2.B+SGV)';
   err[2154].alarm[1] := WSTRING#'PLC - Verstellung Scanner nicht referenziert, händisch neu referenzieren (-8M1.B+SGV)';
   err[2154].alarm[2] := WSTRING#'PLC - adjustment scannerhousing reference not ok, reference manualy (-8M1.B+SGV)';
   err[2154].alarm[3] := WSTRING#'PLC - posizionamento scanner riferimento non coretto, fare corsa di riferimento (-8M1.B+SGV)';
   err[2154].alarm[4] := WSTRING#'PLC - positionnement de scanner référence non correcte, manuel de référence (-8M1.B+SGV)';
   err[2154].alarm[5] := WSTRING#'PLC - el ajuste de del escáner referencia no ok, manual de referencia (-8M1.B+SGV)';
   err[2155].alarm[1] := WSTRING#'PLC - Verstellung Scanner Referenzfahrt aktiv  (-8M1.B+SGV)';
   err[2155].alarm[2] := WSTRING#'PLC - adjustment scannerhousing reference run active (-8M1.B+SGV)';
   err[2155].alarm[3] := WSTRING#'PLC - posizionamento scanner corsa di riferimento attiva (-8M1.B+SGV)';
   err[2155].alarm[4] := WSTRING#'PLC - positionnement de scanner exécution de référence active (-8M1.B+SGV)';
   err[2155].alarm[5] := WSTRING#'PLC - el ajuste de del escáner ejecución de referencia activa (-8M1.B+SGV)';
   err[2156].alarm[1] := WSTRING#'PLC - Verstellung Scanner nicht in Position (-8M1.B+SGV)';
   err[2156].alarm[2] := WSTRING#'PLC - adjustment scannerhousing not in position (-8M1.B+SGV)';
   err[2156].alarm[3] := WSTRING#'PLC - posizionamento scanner non in posizione (-8M1.B+SGV)';
   err[2156].alarm[4] := WSTRING#'PLC - positionnement de scanner pas en position (-8M1.B+SGV)';
   err[2156].alarm[5] := WSTRING#'PLC - el ajuste de del escáner no está en posición (-8M1.B+SGV)';
   err[2157].alarm[1] := WSTRING#'PLC - Verstellung Scanner am Pc auf Hand geschalten (-8M1.B+SGV)';
   err[2157].alarm[2] := WSTRING#'PLC - adjustment scannerhousing set on manual mode on Pc (-8M1.B+SGV)';
   err[2157].alarm[3] := WSTRING#'PLC - posizionamento scanner attivata modalità manuale sul Pc (-8M1.B+SGV)';
   err[2157].alarm[4] := WSTRING#'PLC - positionnement de scanner passé en mode manuel sur le Pc (-8M1.B+SGV)';
   err[2157].alarm[5] := WSTRING#'PLC - el ajuste de del escáner cambiado a manual en la Pc (-8M1.B+SGV)';
   err[2160].alarm[1] := WSTRING#'PLC - Störung Verstellung Messbalken oben (-8M1.T+SGV)';
   err[2160].alarm[2] := WSTRING#'PLC - fault adjustment metering bar top (-8M1.T+SGV)';
   err[2160].alarm[3] := WSTRING#'PLC - errore posizionamento barra di misura superiore (-8M1.T+SGV)';
   err[2160].alarm[4] := WSTRING#'PLC - défaut positionnement de barre de mesure supérieure (-8M1.T+SGV)';
   err[2160].alarm[5] := WSTRING#'PLC - fallo el ajuste de barra de medición superior (-8M1.T+SGV)';
   err[2160].alarm[6..8] := WSTRING#'';
   err[2161].alarm[1] := WSTRING#'PLC - Störung Encoder - Verstellung Messbalken oben (-8B1.T+SGV)';
   err[2161].alarm[2] := WSTRING#'PLC - fault encoder - adjustment metering bar top (-8B1.T+SGV)';
   err[2161].alarm[3] := WSTRING#'PLC - errore encoder - posizionamento barra di misura superiore (-8B1.T+SGV)';
   err[2161].alarm[4] := WSTRING#'PLC - défaut codeur - positionnement de barre de mesure supérieure (-8B1.T+SGV)';
   err[2161].alarm[5] := WSTRING#'PLC - fallo codificador - el ajuste de barra de medición superior (-8B1.T+SGV)';
   err[2161].alarm[6..8] := WSTRING#'';
   err[2162].alarm[1] := WSTRING#'PLC - Störung Sensor Endstellung links - Verstellung Messbalken oben (-8S1.T+SGV)';
   err[2162].alarm[2] := WSTRING#'PLC - fault sensor limit switch position left - adjustment metering bar top (-8S1.T+SGV)';
   err[2162].alarm[3] := WSTRING#'PLC - errore sensore posizione sinistra - posizionamento barra di misura superiore (-8S1.T+SGV)';
   err[2162].alarm[4] := WSTRING#'PLC - défaut capteur position du fin de course à gauche - positionnement de barre de mesure supérieure (-8S1.T+SGV)';
   err[2162].alarm[5] := WSTRING#'PLC - fallo sensor posición de límite a la izquierda - el ajuste de barra de medición superior (-8S1.T+SGV)';
   err[2162].alarm[6..8] := WSTRING#'';
   err[2163].alarm[1] := WSTRING#'PLC - Störung Sensor Endstellung rechts - Verstellung Messbalken oben (-8S2.T+SGV)';
   err[2163].alarm[2] := WSTRING#'PLC - fault sensor limit switch position right - adjustment metering bar top (-8S2.T+SGV)';
   err[2163].alarm[3] := WSTRING#'PLC - errore sensore posizione destra - posizionamento barra di misura superiore (-8S2.T+SGV)';
   err[2163].alarm[4] := WSTRING#'PLC - défaut capteur position du fin de course à droite - positionnement de barre de mesure supérieure (-8S2.T+SGV)';
   err[2163].alarm[5] := WSTRING#'PLC - fallo sensor posición de límite a la derecha - el ajuste de barra de medición superior (-8S2.T+SGV)';
   err[2163].alarm[6..8] := WSTRING#'';
   err[2164].alarm[1] := WSTRING#'PLC - Verstellung Messbalken oben nicht referenziert, händisch neu referenzieren (-8M1.T+SGV)';
   err[2164].alarm[2] := WSTRING#'PLC - adjustment metering bar top reference not ok, reference manualy (-8M1.T+SGV)';
   err[2164].alarm[3] := WSTRING#'PLC - posizionamento barra di misura superiore riferimento non coretto, fare corsa di riferimento (-8M1.T+SGV)';
   err[2164].alarm[4] := WSTRING#'PLC - positionnement de barre de mesure supérieure référence non correcte, manuel de référence (-8M1.T+SGV)';
   err[2164].alarm[5] := WSTRING#'PLC - el ajuste de barra de medición superior referencia no ok, manual de referencia (-8M1.T+SGV)';
   err[2164].alarm[6..8] := WSTRING#'';
   err[2165].alarm[1] := WSTRING#'PLC - Verstellung Messbalken oben Referenzfahrt aktiv  (-8M1.T+SGV)';
   err[2165].alarm[2] := WSTRING#'PLC - adjustment metering bar top reference run active (-8M1.T+SGV)';
   err[2165].alarm[3] := WSTRING#'PLC - posizionamento barra di misura superiore corsa di riferimento attiva (-8M1.T+SGV)';
   err[2165].alarm[4] := WSTRING#'PLC - positionnement de barre de mesure supérieure exécution de référence active (-8M1.T+SGV)';
   err[2165].alarm[5] := WSTRING#'PLC - el ajuste de barra de medición superior ejecución de referencia activa (-8M1.T+SGV)';
   err[2165].alarm[6..8] := WSTRING#'';
   err[2166].alarm[1] := WSTRING#'PLC - Verstellung Messbalken oben nicht in Position (-8M1.T+SGV)';
   err[2166].alarm[2] := WSTRING#'PLC - adjustment metering bar top not in position (-8M1.T+SGV)';
   err[2166].alarm[3] := WSTRING#'PLC - posizionamento barra di misura superiore non in posizione (-8M1.T+SGV)';
   err[2166].alarm[4] := WSTRING#'PLC - positionnement de barre de mesure supérieure pas en position (-8M1.T+SGV)';
   err[2166].alarm[5] := WSTRING#'PLC - el ajuste de barra de medición superior no está en posición (-8M1.T+SGV)';
   err[2166].alarm[6..8] := WSTRING#'';
   err[2167].alarm[1] := WSTRING#'PLC - Verstellung Messbalken oben am Pc auf Hand geschalten (-8M1.T+SGV)';
   err[2167].alarm[2] := WSTRING#'PLC - adjustment metering bar top set on manual mode on Pc (-8M1.T+SGV)';
   err[2167].alarm[3] := WSTRING#'PLC - posizionamento barra di misura superiore attivata modalità manuale sul Pc (-8M1.T+SGV)';
   err[2167].alarm[4] := WSTRING#'PLC - positionnement de barre de mesure supérieure passé en mode manuel sur le Pc (-8M1.T+SGV)';
   err[2167].alarm[5] := WSTRING#'PLC - el ajuste de barra de medición superior cambiado a manual en la Pc (-8M1.T+SGV)';
   err[2170].alarm[1] := WSTRING#'PLC - Störung Verstellung Messbalken links (-8M1.L+SGV)';
   err[2170].alarm[2] := WSTRING#'PLC - fault adjustment metering bar left (-8M1.L+SGV)';
   err[2170].alarm[3] := WSTRING#'PLC - errore posizionamento barra di misura di sinistra (-8M1.L+SGV)';
   err[2170].alarm[4] := WSTRING#'PLC - défaut positionnement de barre de mesure gauche (-8M1.L+SGV)';
   err[2170].alarm[5] := WSTRING#'PLC - fallo el ajuste de barra de medición izquierda (-8M1.L+SGV)';
   err[2170].alarm[6..8] := WSTRING#'';
   err[2171].alarm[1] := WSTRING#'PLC - Störung Encoder - Verstellung Messbalken links (-8B1.L+SGV)';
   err[2171].alarm[2] := WSTRING#'PLC - fault encoder - adjustment metering bar left (-8B1.L+SGV)';
   err[2171].alarm[3] := WSTRING#'PLC - errore encoder - posizionamento barra di misura di sinistra (-8B1.L+SGV)';
   err[2171].alarm[4] := WSTRING#'PLC - défaut codeur - positionnement de barre de mesure gauche (-8B1.L+SGV)';
   err[2171].alarm[5] := WSTRING#'PLC - fallo codificador - el ajuste de barra de medición izquierda (-8B1.L+SGV)';
   err[2171].alarm[6..8] := WSTRING#'';
   err[2172].alarm[1] := WSTRING#'PLC - Störung Sensor Endstellung links - Verstellung Messbalken links (-8S1.L+SGV)';
   err[2172].alarm[2] := WSTRING#'PLC - fault sensor limit switch position left - adjustment metering bar left (-8S1.L+SGV)';
   err[2172].alarm[3] := WSTRING#'PLC - errore sensore posizione sinistra - posizionamento barra di misura di sinistra (-8S1.L+SGV)';
   err[2172].alarm[4] := WSTRING#'PLC - défaut capteur position du fin de course à gauche - positionnement de barre de mesure gauche (-8S1.L+SGV)';
   err[2172].alarm[5] := WSTRING#'PLC - fallo sensor posición de límite a la izquierda - el ajuste de barra de medición izquierda (-8S1.L+SGV)';
   err[2172].alarm[6..8] := WSTRING#'';
   err[2173].alarm[1] := WSTRING#'PLC - Störung Sensor Endstellung rechts - Verstellung Messbalken links (-8S2.L+SGV)';
   err[2173].alarm[2] := WSTRING#'PLC - fault sensor limit switch position right - adjustment metering bar left (-8S2.L+SGV)';
   err[2173].alarm[3] := WSTRING#'PLC - errore sensore posizione destra - posizionamento barra di misura di sinistra (-8S2.L+SGV)';
   err[2173].alarm[4] := WSTRING#'PLC - défaut capteur position du fin de course à droite - positionnement de barre de mesure gauche (-8S2.L+SGV)';
   err[2173].alarm[5] := WSTRING#'PLC - fallo sensor posición de límite a la derecha - el ajuste de barra de medición izquierda (-8S2.L+SGV)';
   err[2173].alarm[6..8] := WSTRING#'';
   err[2174].alarm[1] := WSTRING#'PLC - Verstellung Messbalken links nicht referenziert, händisch neu referenzieren (-8M1.L+SGV)';
   err[2174].alarm[2] := WSTRING#'PLC - adjustment metering bar left reference not ok, reference manualy (-8M1.L+SGV)';
   err[2174].alarm[3] := WSTRING#'PLC - posizionamento barra di misura di sinistra riferimento non coretto, fare corsa di riferimento (-8M1.L+SGV)';
   err[2174].alarm[4] := WSTRING#'PLC - positionnement de barre de mesure gauche référence non correcte, manuel de référence (-8M1.L+SGV)';
   err[2174].alarm[5] := WSTRING#'PLC - el ajuste de barra de medición izquierda referencia no ok, manual de referencia (-8M1.L+SGV)';
   err[2174].alarm[6..8] := WSTRING#'';
   err[2175].alarm[1] := WSTRING#'PLC - Verstellung Messbalken links Referenzfahrt aktiv  (-8M1.L+SGV)';
   err[2175].alarm[2] := WSTRING#'PLC - adjustment metering bar left reference run active (-8M1.L+SGV)';
   err[2175].alarm[3] := WSTRING#'PLC - posizionamento barra di misura di sinistra corsa di riferimento attiva (-8M1.L+SGV)';
   err[2175].alarm[4] := WSTRING#'PLC - positionnement de barre de mesure gauche exécution de référence active (-8M1.L+SGV)';
   err[2175].alarm[5] := WSTRING#'PLC - el ajuste de barra de medición izquierda ejecución de referencia activa (-8M1.L+SGV)';
   err[2175].alarm[6..8] := WSTRING#'';
   err[2176].alarm[1] := WSTRING#'PLC - Verstellung Messbalken links nicht in Position (-8M1.L+SGV)';
   err[2176].alarm[2] := WSTRING#'PLC - adjustment metering bar left not in position (-8M1.L+SGV)';
   err[2176].alarm[3] := WSTRING#'PLC - posizionamento barra di misura di sinistra non in posizione (-8M1.L+SGV)';
   err[2176].alarm[4] := WSTRING#'PLC - positionnement de barre de mesure gauche pas en position (-8M1.L+SGV)';
   err[2176].alarm[5] := WSTRING#'PLC - el ajuste de barra de medición izquierda no está en posición (-8M1.L+SGV)';
   err[2176].alarm[6..8] := WSTRING#'';
   err[2177].alarm[1] := WSTRING#'PLC - Verstellung Messbalken links am Pc auf Hand geschalten (-8M1.L+SGV)';
   err[2177].alarm[2] := WSTRING#'PLC - adjustment metering bar left set on manual mode on Pc (-8M1.L+SGV)';
   err[2177].alarm[3] := WSTRING#'PLC - posizionamento barra di misura di sinistra attivata modalità manuale sul Pc (-8M1.L+SGV)';
   err[2177].alarm[4] := WSTRING#'PLC - positionnement de barre de mesure gauche passé en mode manuel sur le Pc (-8M1.L+SGV)';
   err[2177].alarm[5] := WSTRING#'PLC - el ajuste de barra de medición izquierda cambiado a manual en la Pc (-8M1.L+SGV)';
   err[2177].alarm[6..8] := WSTRING#'';
   err[2180].alarm[1] := WSTRING#'PLC - Störung Verstellung Messbalken rechts (-8M1.R+SGV)';
   err[2180].alarm[2] := WSTRING#'PLC - fault adjustment metering bar right (-8M1.R+SGV)';
   err[2180].alarm[3] := WSTRING#'PLC - errore posizionamento barra di misura di destra (-8M1.R+SGV)';
   err[2180].alarm[4] := WSTRING#'PLC - défaut positionnement de barre de mesure à droite (-8M1.R+SGV)';
   err[2180].alarm[5] := WSTRING#'PLC - fallo el ajuste de barra de medición derecha (-8M1.R+SGV)';
   err[2180].alarm[6..8] := WSTRING#'';
   err[2181].alarm[1] := WSTRING#'PLC - Störung Encoder - Verstellung Messbalken rechts (-8B1.R+SGV)';
   err[2181].alarm[2] := WSTRING#'PLC - fault encoder - adjustment metering bar right (-8B1.R+SGV)';
   err[2181].alarm[3] := WSTRING#'PLC - errore encoder - posizionamento barra di misura di destra (-8B1.R+SGV)';
   err[2181].alarm[4] := WSTRING#'PLC - défaut codeur - positionnement de barre de mesure à droite (-8B1.R+SGV)';
   err[2181].alarm[5] := WSTRING#'PLC - fallo codificador - el ajuste de barra de medición derecha (-8B1.R+SGV)';
   err[2181].alarm[6..8] := WSTRING#'';
   err[2182].alarm[1] := WSTRING#'PLC - Störung Sensor Endstellung links - Verstellung Messbalken rechts (-8S1.R+SGV)';
   err[2182].alarm[2] := WSTRING#'PLC - fault sensor limit switch position left - adjustment metering bar right (-8S1.R+SGV)';
   err[2182].alarm[3] := WSTRING#'PLC - errore sensore posizione sinistra - posizionamento barra di misura di destra (-8S1.R+SGV)';
   err[2182].alarm[4] := WSTRING#'PLC - défaut capteur position du fin de course à gauche - positionnement de barre de mesure à droite (-8S1.R+SGV)';
   err[2182].alarm[5] := WSTRING#'PLC - fallo sensor posición de límite a la izquierda - el ajuste de barra de medición derecha (-8S1.R+SGV)';
   err[2182].alarm[6..8] := WSTRING#'';
   err[2183].alarm[1] := WSTRING#'PLC - Störung Sensor Endstellung rechts - Verstellung Messbalken rechts (-8S2.R+SGV)';
   err[2183].alarm[2] := WSTRING#'PLC - fault sensor limit switch position right - adjustment metering bar right (-8S2.R+SGV)';
   err[2183].alarm[3] := WSTRING#'PLC - errore sensore posizione destra - posizionamento barra di misura di destra (-8S2.R+SGV)';
   err[2183].alarm[4] := WSTRING#'PLC - défaut capteur position du fin de course à droite - positionnement de barre de mesure à droite (-8S2.R+SGV)';
   err[2183].alarm[5] := WSTRING#'PLC - fallo sensor posición de límite a la derecha - el ajuste de barra de medición derecha (-8S2.R+SGV)';
   err[2183].alarm[6..8] := WSTRING#'';
   err[2184].alarm[1] := WSTRING#'PLC - Verstellung Messbalken rechts nicht referenziert, händisch neu referenzieren (-8M1.R+SGV)';
   err[2184].alarm[2] := WSTRING#'PLC - adjustment metering bar right reference not ok, reference manualy (-8M1.R+SGV)';
   err[2184].alarm[3] := WSTRING#'PLC - posizionamento barra di misura di destra riferimento non coretto, fare corsa di riferimento (-8M1.R+SGV)';
   err[2184].alarm[4] := WSTRING#'PLC - positionnement de barre de mesure à droite référence non correcte, manuel de référence (-8M1.R+SGV)';
   err[2184].alarm[5] := WSTRING#'PLC - el ajuste de barra de medición derecha referencia no ok, manual de referencia (-8M1.R+SGV)';
   err[2184].alarm[6..8] := WSTRING#'';
   err[2185].alarm[1] := WSTRING#'PLC - Verstellung Messbalken rechts Referenzfahrt aktiv  (-8M1.R+SGV)';
   err[2185].alarm[2] := WSTRING#'PLC - adjustment metering bar right reference run active (-8M1.R+SGV)';
   err[2185].alarm[3] := WSTRING#'PLC - posizionamento barra di misura di destra corsa di riferimento attiva (-8M1.R+SGV)';
   err[2185].alarm[4] := WSTRING#'PLC - positionnement de barre de mesure à droite exécution de référence active (-8M1.R+SGV)';
   err[2185].alarm[5] := WSTRING#'PLC - el ajuste de barra de medición derecha ejecución de referencia activa (-8M1.R+SGV)';
   err[2185].alarm[6..8] := WSTRING#'';
   err[2186].alarm[1] := WSTRING#'PLC - Verstellung Messbalken rechts nicht in Position (-8M1.R+SGV)';
   err[2186].alarm[2] := WSTRING#'PLC - adjustment metering bar right not in position (-8M1.R+SGV)';
   err[2186].alarm[3] := WSTRING#'PLC - posizionamento barra di misura di destra non in posizione (-8M1.R+SGV)';
   err[2186].alarm[4] := WSTRING#'PLC - positionnement de barre de mesure à droite pas en position (-8M1.R+SGV)';
   err[2186].alarm[5] := WSTRING#'PLC - el ajuste de barra de medición derecha no está en posición (-8M1.R+SGV)';
   err[2186].alarm[6..8] := WSTRING#'';
   err[2187].alarm[1] := WSTRING#'PLC - Verstellung Messbalken rechts am Pc auf Hand geschalten (-8M1.R+SGV)';
   err[2187].alarm[2] := WSTRING#'PLC - adjustment metering bar right set on manual mode on Pc (-8M1.R+SGV)';
   err[2187].alarm[3] := WSTRING#'PLC - posizionamento barra di misura di destra attivata modalità manuale sul Pc (-8M1.R+SGV)';
   err[2187].alarm[4] := WSTRING#'PLC - positionnement de barre de mesure à droite passé en mode manuel sur le Pc (-8M1.R+SGV)';
   err[2187].alarm[5] := WSTRING#'PLC - el ajuste de barra de medición derecha cambiado a manual en la Pc (-8M1.R+SGV)';
   err[2187].alarm[6..8] := WSTRING#'';
   err[2190].alarm[1] := WSTRING#'PLC - Störung Sensor für Distanzmessung von oben (-8B1+SGV)';
   err[2190].alarm[2] := WSTRING#'PLC - fault sensor distance measurement from top (-8B1+SGV)';
   err[2190].alarm[3] := WSTRING#'PLC - errore sensore misurazione della distanza dall`alto(-8B1+SGV)';
   err[2190].alarm[4] := WSTRING#'PLC - défaut capteur mesure de distance en haut (-8B1+SGV)';
   err[2190].alarm[5] := WSTRING#'PLC - fallo de sensor medición de distancia del sensor superior (-8B1+SGV)';
   err[2191].alarm[1] := WSTRING#'PLC - Störung Sensor für Distanzmessung von links (-8B2+SGV)';
   err[2191].alarm[2] := WSTRING#'PLC - fault sensor distance measurement from left (-8B2+SGV)';
   err[2191].alarm[3] := WSTRING#'PLC - errore sensore misurazione della distanza da sinistra (-8B2+SGV)';
   err[2191].alarm[4] := WSTRING#'PLC - défaut capteur mesure de distance de gauche à droite (-8B2+SGV)';
   err[2191].alarm[5] := WSTRING#'PLC - fallo de sensor medición de distancia del sensor desde la izquierda (-8B2+SGV)';
   err[2192].alarm[1] := WSTRING#'PLC - Störung Sensor für Distanzmessung von rechts (-8B3+SGV)';
   err[2192].alarm[2] := WSTRING#'PLC - fault sensor distance measurement from right (-8B3+SGV)';
   err[2192].alarm[3] := WSTRING#'PLC - errore sensore misurazione della distanza da destra (-8B3+SGV)';
   err[2192].alarm[4] := WSTRING#'PLC - défaut capteur mesure de distance de droite à gauche (-8B3+SGV)';
   err[2192].alarm[5] := WSTRING#'PLC - fallo de sensor medición de distancia del sensor desde la derecha (-8B3+SGV)';
   err[2200].alarm[1] := WSTRING#'PLC - Störung Profinet Slave LINMOT Servodrive - Verstellung Messbalken oben (-8U1.T+SGV)';
   err[2200].alarm[2] := WSTRING#'PLC - fault profinet-slave LINMOT Servodrive - adjustment metering bar top (-8U1.T+SGV)';
   err[2200].alarm[3] := WSTRING#'PLC - profinet-slave LINMOT Servodrive - posizionamento barra di misura superiore (-8U1.T+SGV)';
   err[2200].alarm[4] := WSTRING#'PLC - profinet-slave LINMOT Servodrive - positionnement de barre de mesure supérieure (-8U1.T+SGV)';
   err[2200].alarm[5] := WSTRING#'PLC - profinet-slave LINMOT Servodrive - el ajuste de barra de medición superior (-8U1.T+SGV)';
   err[2201].alarm[1] := WSTRING#'PLC - Störung Profinet Slave LINMOT Servodrive - Verstellung Messbalken links (-8U1.L+SGV)';
   err[2201].alarm[2] := WSTRING#'PLC - fault profinet-slave LINMOT Servodrive - adjustment metering bar left (-8U1.L+SGV)';
   err[2201].alarm[3] := WSTRING#'PLC - profinet-slave LINMOT Servodrive - posizionamento barra di misura di sinistra (-8U1.L+SGV)';
   err[2201].alarm[4] := WSTRING#'PLC - profinet-slave LINMOT Servodrive - positionnement de barre de mesure gauche (-8U1.L+SGV)';
   err[2201].alarm[5] := WSTRING#'PLC - profinet-slave LINMOT Servodrive - el ajuste de barra de medición izquierda (-8U1.L+SGV)';
   err[2202].alarm[1] := WSTRING#'PLC - Störung Profinet Slave LINMOT Servodrive - Verstellung Messbalken rechts (-8U1.R+SGV)';
   err[2202].alarm[2] := WSTRING#'PLC - fault profinet-slave LINMOT Servodrive - adjustment metering bar right (-8U1.R+SGV)';
   err[2202].alarm[3] := WSTRING#'PLC - profinet-slave LINMOT Servodrive - posizionamento barra di misura di destra(-8U1.R+SGV)';
   err[2202].alarm[4] := WSTRING#'PLC - profinet-slave LINMOT Servodrive - positionnement de barre de mesure à droite (-8U1.R+SGV)';
   err[2202].alarm[5] := WSTRING#'PLC - profinet-slave LINMOT Servodrive - el ajuste de barra de medición derecha (-8U1.R+SGV)';
END_DATA_BLOCK

DATA_BLOCK "G"   // DB350
{ S7_Optimized_Access := 'TRUE' }
// stored: AutoNumber false, IsRetainMemResEnabled true, MemoryReserve 100, RetainMemoryReserve 100
   VAR RETAIN
      lampTest : Bool;   // lamp test
      settingMode : Bool;   // setting mode active
      jogMode : Bool;   // jog mode active
      scannerReady : Bool;   // scanner ready
      scannerErr : Bool;   // scanner error
      scannerEmpty : Bool;   // scanner empty
      releaseInfeed : Bool;   // release infeed
      auto : Bool;   // automatic mode adjustment
      ack : Bool;   // reset faults general
      ackPC : Bool;   // reset faults pc
      err : Bool;   // fault general
      war : Bool;   // warning general
      info : Bool;   // info general
      pneOk : Bool;   // pneumatic ok
      comOk : Bool;   // communication ok
      "errPs-0F1.1+SGV" : Bool;   // fault voltage monitoring for power supply
      "errAc-0E1+SGV" : Bool;   // fault air conditioner 1 visual
      "errAc-0E2+SGX" : Bool;   // fault air conditioner Xray
      "errAc-0E1.1+SGV" : Bool;   // fault air conditioner 2 visual
      errComPc : Bool;   // fault communication with pc
      errProfinet : Bool;   // fault profinet
      errAdjScanner : Bool;   // fault adjustment scanner
      errAdjTop : Bool;   // fault adjustment top
      errAdjLeft : Bool;   // fault adjustment left
      errAdjRight : Bool;   // fault adjustment right
      errVersion : Bool;   // fault version
      errSafetyModules : Bool;   // fault safety modules
      errNoReleaseInf : Bool;   // fault no release from plc to infeed
      Batch : Struct   // batch info - board data
         stdActive : Bool;   // standardisation batch active
         width : Real;   // board width [mm]
         widthMin : Real;   // board width min [mm]
         widthMax : Real;   // board width max [mm]
         thickness : Real;   // board thickness [mm]
         thicknessMin : Real;   // board thickness min [mm]
         thicknessMax : Real;   // board thickness max [mm]
         widthMeasure : Real;   // board width measured value from sensors [mm]
         thicknessMeasure : Real;   // board thickness measured value from sensor [mm]
         senLeftVal : Real;   // sensor left value [mm]
         senRightVal : Real;   // sensor right value [mm]
         offsetBoard { ExternalWritable := 'False'} : Real;   // offset board to middle [mm] - bigger then zero then board is shifted to the left side
      END_STRUCT;
      Cfg : Struct   // config
         adjScannerActive : Bool;   // adjustment scanner housing active
         adjTopActive : Bool;   // adjustment camera top active
         adjLeftActive : Bool;   // adjustment camera left active
         adjRightActive : Bool;   // adjustment camera right active
         adjTopActiveLinMot : Bool;   // adjustment top active - linear drive
         adjLeftActiveLinMot : Bool;   // adjustment left active - linear drive
         adjRightActiveLinMot : Bool;   // adjustment right active - linear drive
         xrayActive : Bool;   // xray active
         enc1Active : Bool;   // encoder 1 active (infeed)
         senTopActive : Bool;   // sensor top active for random adjustment
         senLeftActive : Bool;   // sensor left active for random adjustment
         senRightActive : Bool;   // sensor right active for random adjustment
         modeBoardPassing : Int;   // 1=left / 2=right / 3=middle
         modeDimension : Int;   // 1=fixed / 2=random width / 3=random thickness / 4=random width + thickness
         modeRandomAdj : Int;   // 1=with sensor / 2=with external data
         enc1Gain : Real;   // encoder 1 gain (infeed)
      END_STRUCT;
      adjScannerOff : Bool;   // adjustment scanner housing off (only manual movement possible )
      adjTopOff : Bool;   // adjustment camera top off (only manual movement possible )
      adjLeftOff : Bool;   // adjustment camera left off (only manual movement possible )
      adjRightOff : Bool;   // adjustment camera right off (only manual movement possible )
   END_VAR
   VAR
      air1Off { ExternalAccessible := 'False'; ExternalVisible := 'False'; ExternalWritable := 'False'} : Bool;
      air2Off { ExternalAccessible := 'False'; ExternalVisible := 'False'; ExternalWritable := 'False'} : Bool;
      airXrayOff { ExternalAccessible := 'False'; ExternalVisible := 'False'; ExternalWritable := 'False'} : Bool;
      airDehOff { ExternalAccessible := 'False'; ExternalVisible := 'False'; ExternalWritable := 'False'} : Bool;
   END_VAR
BEGIN
END_DATA_BLOCK

DATA_BLOCK "Mot"   // DB322
{ S7_Optimized_Access := 'TRUE' }
// stored: AutoNumber false, IsRetainMemResEnabled true, MemoryReserve 500, RetainMemoryReserve 500
   VAR RETAIN
      "8M1.B" : "TypeMotor";   // adjustment scanner
      "8M1.T" : "TypeMotor";   // adjustment top - normal drive
      "8M1.L" : "TypeMotor";   // adjustment left - normal drive
      "8M1.R" : "TypeMotor";   // adjustment right - normal drive
      "8U1.T" : "TypeMotor";   // adjustment top - linear drive
      "8U1.L" : "TypeMotor";   // adjustment left - linear drive
      "8U1.R" : "TypeMotor";   // adjustment right - linear drive
   END_VAR
BEGIN
   "8M1.B".description := WSTRING#'Motor Aufgabeförderer 1 - Zubringung';
   "8M1.T".description := WSTRING#'Motor Aufgabeförderer 2 - Zubringung';
   "8M1.L".description := WSTRING#'Motor Zerteiler - Zubringung';
   "8M1.R".description := WSTRING#'Motor Überbrückungsförderer - Zubringung';
   "8U1.T".description := WSTRING#'Motor Aufgabeförderer 2 - Zubringung';
   "8U1.L".description := WSTRING#'Motor Zerteiler - Zubringung';
   "8U1.R".description := WSTRING#'Motor Überbrückungsförderer - Zubringung';
END_DATA_BLOCK

DATA_BLOCK "Param"   // DB352
{ S7_Optimized_Access := 'FALSE' }
// stored: AutoNumber false
   VAR RETAIN
      Plc : "TypeHeaderPlc";   // Header Plc
      Rd : Struct
         watchdog : Int := 0;   // watchdog
         adjHousingOff : Int := 0;   // adjustment scanner housing off (only manual movement possible ) [On/Off]
         adjTopOff : Int := 0;   // adjustment camera top off (only manual movement possible ) [On/Off]
         adjLeftOff : Int := 0;   // adjustment camera left off (only manual movement possible ) [On/Off]
         adjRightOff : Int := 0;   // adjustment camera right off (only manual movement possible ) [On/Off]
         adjLaserTopLeftStepMotOff : Int;   // adjustment laser top left off (only manual movement possible ) [On/Off]
         adjLaserTopRightStepMotOff : Int;   // adjustment laser top right off (only manual movement possible ) [On/Off]
         adjLaserLeftTopStepMotOff : Int;   // adjustment laser left top off (only manual movement possible ) [On/Off]
         adjLaserLeftBottomStepMotOff : Int;   // adjustment laser left bottom off (only manual movement possible ) [On/Off]
         adjLaserRightTopStepMotOff : Int;   // adjustment laser right top off (only manual movement possible ) [On/Off]
         adjLaserRightBottomStepMotOff : Int;   // adjustment laser right bottom off (only manual movement possible ) [On/Off]
         param1 : Int;
         param2 : Int;
         param3 : Int;
         param4 : Int;
         air1Off : Int := 0;   // air conditioner 1 scannerhousing visual measurement [On/Off]
         air2Off : Int := 0;   // air conditioner 2 scannerhousing visual measurement [On/Off]
         airXrayOff : Int := 0;   // air conditioner scannerhousing x-ray measurement [On/Off]
         airDehOff : Int := 0;   // air dehumidifier
         param5 : Int := 0;
         param6 : Int := 0;
         blowOffImpuls : Int := 400;   // blow off impulse [ms]
         blowOffIbreak : Int := 400;   // blow off minimum break to start new cycle [ms]
         blowOffintervall : Int := 120;   // blow off interval if no board pass [s]
         param10 : Int := 0;
         air1Active : Int := 1;   // air conditioner 1 scannerhousing visual measurement active [On/Off]
         air1InputNo : Int := 0;   // air conditioner 1 scannerhousing visual measurement input normal [On/Off]
         air2Active : Int := 0;   // air conditioner 2 scannerhousing visual measurement active [On/Off]
         air2InputNo : Int := 0;   // air conditioner 2 scannerhousing visual measurement input normal [On/Off]
         airXrayActive : Int := 1;   // air conditioner scannerhousing x-ray measurement active [On/Off]
         airXrayInputNo : Int := 0;   // air conditioner scannerhousing x-ray measurement input normal [On/Off]
         airDehActive : Int := 0;   // air dehumidifier active [On/Off]
         airDehInputNo : Int := 0;   // air dehumidifier input normal open [On/Off]
         param11 : Int := 0;
         blowOffintervallOff : Int := 600;   // blow off interval if no board pass switches off after this time [s]
         blowOffDelayStartBottom : Int := 0;   // blow off delay start for valve bottom [ms]
         blowOffDelayStartLeft : Int := 0;   // blow off delay start for valve left [ms]
         blowOffDelayStartRight : Int := 0;   // blow off delay start for valve right [ms]
         blowOffDelayStartXray : Int := 0;   // blow off delay start for valve xray [ms]
         blowOffImpulsBottom : Int := 400;   // blow off impulse for valve bottom [ms]
         blowOffImpulsLeft : Int := 400;   // blow off impulse for valve left [ms]
         blowOffImpulsRight : Int := 400;   // blow off impulse for valve right [ms]
         blowOffImpulsXray : Int := 400;   // blow off impulse for valve xray [ms]
         ParamRes : Array[1..58] of Int;
      END_STRUCT;
   END_VAR
BEGIN
   Plc.conActive := FALSE;
   Plc.err := FALSE;
   Plc.errWd := FALSE;
   Plc.errSd := FALSE;
   Plc.errRd := FALSE;
   Plc.bit05 := FALSE;
   Plc.bit06 := FALSE;
   Plc.bit07 := FALSE;
   Plc.sdBusy := FALSE;
   Plc.sdDone := FALSE;
   Plc.rdBusy := FALSE;
   Plc.rdDone := FALSE;
   Plc.sdOverload := FALSE;
   Plc.statistic := FALSE;
   Plc.bit16 := FALSE;
   Plc.bit17 := FALSE;
   Plc.sdState := 16#0000;
   Plc.sdLastErrState := 16#0000;
   Plc.sdLenght := 0;
   Plc.sdCps := 0;
   Plc.rdState := 16#0000;
   Plc.rdLastErrState := 16#0000;
   Plc.rdLenght := 0;
   Plc.rdCps := 0;
   Plc.in18 := 0;
   Rd.ParamRes[1..50] := 0;
END_DATA_BLOCK

DATA_BLOCK "Sen"   // DB324
{ S7_Optimized_Access := 'TRUE' }
// stored: AutoNumber false, IsRetainMemResEnabled true, MemoryReserve 500, RetainMemoryReserve 500
   VAR RETAIN
      "1BTR2+SGV" : "TypeSensor";   // light barrier in scannerhousing visual measurement
      "1BTR2+SGX" : "TypeSensor";   // light barrier in scannerhousing x-ray measurement
      "8S1.T" : "TypeSensor";   // adjustment top limit switch innermost position
      "8S2.T" : "TypeSensor";   // adjustment top limit switch outermost position
      "8S1.L" : "TypeSensor";   // adjustment left limit switch innermost position
      "8S2.L" : "TypeSensor";   // adjustment left limit switch outermost position
      "8S1.R" : "TypeSensor";   // adjustment right limit switch innermost position
      "8S2.R" : "TypeSensor";   // adjustment right limit switch outermost position
      "8S1.B" : "TypeSensor";   // adjustment scanner limit switch left position
      "8S2.B" : "TypeSensor";   // adjustment scanner limit switch right position
      "8B1" : "TypeSensor";   // light barrier measuring distance top
      "8B2" : "TypeSensor";   // light barrier measuring distance left
      "8B3" : "TypeSensor";   // light barrier measuring distance right
   END_VAR
BEGIN
   "1BTR2+SGV".description := WSTRING#'Sensor Aufgabförderer 1 Ende belegt - Zubringung';
   "1BTR2+SGX".description := WSTRING#'Sensor Aufgabförderer 2 Ende belegt - Zubringung';
   "8S1.T".description := WSTRING#'Sensor Aufgabförderer 2 Ende belegt - Zubringung';
   "8S2.T".description := WSTRING#'Sensor Aufgabförderer 2 Ende belegt - Zubringung';
   "8S1.L".description := WSTRING#'Sensor Aufgabförderer 2 Ende belegt - Zubringung';
   "8S2.L".description := WSTRING#'Sensor Aufgabförderer 2 Ende belegt - Zubringung';
   "8S1.R".description := WSTRING#'Sensor Aufgabförderer 2 Ende belegt - Zubringung';
   "8S2.R".description := WSTRING#'Sensor Aufgabförderer 2 Ende belegt - Zubringung';
   "8S1.B".description := WSTRING#'Sensor Aufgabförderer 2 Ende belegt - Zubringung';
   "8S2.B".description := WSTRING#'Sensor Aufgabförderer 2 Ende belegt - Zubringung';
END_DATA_BLOCK

DATA_BLOCK "IOLinkConfig"   // DB4000
{ S7_Optimized_Access := 'FALSE' }
// stored: AutoNumber false
   VAR
      "8B1.B" : "TypeIOLinkParamArray";   // sensor IO-Link adjustment scannerhousing
      "8B1" : "TypeIOLinkParamArray";   // sensor IO-Link light barrier measuring distance top
      "8B2" : "TypeIOLinkParamArray";   // sensor IO-Link light barrier measuring distance left
      "8B3" : "TypeIOLinkParamArray";   // sensor IO-Link light barrier measuring distance right
      Empty : "TypeIOLinkParamArray";
      "8B1.B-Restart-Conf" : Bool;   // sensor IO-Link adjustment scannerhousing - restart config
      "8B1-Restart-Conf" : Bool;   // sensor IO-Link light barrier measuring distance top - restart config
      "8B2-Restart-Conf" : Bool;   // sensor IO-Link light barrier measuring distance left - restart config
      "8B3-Restart-Conf" : Bool;   // sensor IO-Link light barrier measuring distance right - restart config
   END_VAR
BEGIN
END_DATA_BLOCK

DATA_BLOCK "Hmi"   // DB75
{ S7_Optimized_Access := 'FALSE'; DB_Accessible_From_OPC_UA := 'FALSE' }
AUTHOR : MICROTEC
FAMILY : HMI
NAME : HMI
VERSION : 1.0
// stored: AutoNumber false, DBAccessibleFromOPCUA false
   VAR RETAIN
      Clock : Struct
         Act : Date_And_Time;
         Tar : Date_And_Time;
         Set : Bool;
         Read : Bool;
      END_STRUCT;
      operatingHours : DInt;   // complete operating hours from Cpu
      TimeOfDay : Time_Of_Day;
      TimeStamp : DTL;
   END_VAR
BEGIN
END_DATA_BLOCK

DATA_BLOCK "AdjFast"   // DB506
{ S7_Optimized_Access := 'TRUE'; DB_Accessible_From_OPC_UA := 'FALSE' }
// stored: AutoNumber false, DBAccessibleFromOPCUA false, MemoryReserve 100
   VAR
      Top { ExternalAccessible := 'False'; ExternalVisible := 'False'; ExternalWritable := 'False'} : Struct   // adjustment top
         Mode : Int := 0;   // 1=VAI / 2=SIN VA / 3=Bestehorn VAJ
         Test : Struct
            ModeActive : Bool := false;   // mode test active (move between testpos 1 and 2)
            TarPos : Real := 5.0;   // target positon [mm]
            TarPos1 : Real := 5.0;   // target positon 1 [mm]
            TarPos2 : Real := 155.0;   // target positon 2 [mm]
            TimePosOk : Time := T#2s;   // time for position ok to switch to other position
         END_STRUCT;
         VAI : Struct
            Par1 : Real := 50.0;   // target positon [mm]
            Par2 : Real := 2.0;   // maximal velocity [m/s]
            Par3 : Real := 12.0;   // acceleration [m/s²]
            Par4 : Real := 12.0;   // deceleration [m/s²]
         END_STRUCT;
         SinVA : Struct
            Par1 : Real := 50.0;   // target positon [mm]
            Par2 : Real := 2.0;   // maximal velocity [m/s]
            Par3 : Real := 18.0;   // maixmal acceleration/deceleration [m/s²]
            Par4 : Real := 0.0;   // not used
         END_STRUCT;
         BestehornVAJ : Struct
            Par1 : Real := 50.0;   // target positon [mm]
            Par2 : Real := 2.0;   // maximal velocity [m/s]
            Par3 : Real := 24.0;   // maixmal acceleration/deceleration [m/s²]
            Par4 : Real := 450.0;   // maximal jerk [m/s³]
         END_STRUCT;
         Current : Struct   // current monitoring
            Man : Struct   // manual mode
               War : Struct
                  MinValue : Real := -3.0;   // min current value
                  MaxValue : Real := 2.0;   // max current value
                  Err : Bool;   // warning error
               END_STRUCT;
               Err : Struct
                  MinValue : Real := -3.0;   // min current value
                  MaxValue : Real := 2.0;   // max current value
                  Err : Bool;   // error
               END_STRUCT;
            END_STRUCT;
            Auto : Struct   // auto mode
               War : Struct
                  MinValue : Real := -15.0;   // min current value
                  MaxValue : Real := 16.0;   // max current value
                  Err : Bool;   // warning error
               END_STRUCT;
               Err : Struct
                  MinValue : Real := -15.0;   // min current value
                  MaxValue : Real := 16.0;   // max current value
                  Err : Bool;   // error
               END_STRUCT;
            END_STRUCT;
         END_STRUCT;
      END_STRUCT;
      Left { ExternalAccessible := 'False'; ExternalVisible := 'False'; ExternalWritable := 'False'} : Struct   // adjustment left
         Mode : Int := 0;   // 1=VAI / 2=SIN VA / 3=Bestehorn VAJ
         Test : Struct
            ModeActive : Bool := false;   // mode test active (move between testpos 1 and 2)
            TarPos : Real := 5.0;   // target positon [mm]
            TarPos1 : Real := 5.0;   // target positon 1 [mm]
            TarPos2 : Real := 155.0;   // target positon 2 [mm]
            TimePosOk : Time := T#2s;   // time for position ok to switch to other position
         END_STRUCT;
         VAI : Struct
            Par1 : Real := 50.0;   // target positon [mm]
            Par2 : Real := 2.0;   // maximal velocity [m/s]
            Par3 : Real := 12.0;   // acceleration [m/s²]
            Par4 : Real := 12.0;   // deceleration [m/s²]
         END_STRUCT;
         SinVA : Struct
            Par1 : Real := 50.0;   // target positon [mm]
            Par2 : Real := 2.0;   // maximal velocity [m/s]
            Par3 : Real := 18.0;   // maixmal acceleration/deceleration [m/s²]
            Par4 : Real := 0.0;   // not used
         END_STRUCT;
         BestehornVAJ : Struct
            Par1 : Real := 50.0;   // target positon [mm]
            Par2 : Real := 2.0;   // maximal velocity [m/s]
            Par3 : Real := 24.0;   // maixmal acceleration/deceleration [m/s²]
            Par4 : Real := 450.0;   // maximal jerk [m/s³]
         END_STRUCT;
         Current : Struct   // current monitoring
            Man : Struct   // manual mode
               War : Struct
                  MinValue : Real := -3.0;   // min current value
                  MaxValue : Real := 2.0;   // max current value
                  Err : Bool;   // warning error
               END_STRUCT;
               Err : Struct
                  MinValue : Real := -3.0;   // min current value
                  MaxValue : Real := 2.0;   // max current value
                  Err : Bool;   // error
               END_STRUCT;
            END_STRUCT;
            Auto : Struct   // auto mode
               War : Struct
                  MinValue : Real := -15.0;   // min current value
                  MaxValue : Real := 16.0;   // max current value
                  Err : Bool;   // warning error
               END_STRUCT;
               Err : Struct
                  MinValue : Real := -15.0;   // min current value
                  MaxValue : Real := 16.0;   // max current value
                  Err : Bool;   // error
               END_STRUCT;
            END_STRUCT;
         END_STRUCT;
      END_STRUCT;
      Right { ExternalAccessible := 'False'; ExternalVisible := 'False'; ExternalWritable := 'False'} : Struct   // adjustment right
         Mode : Int := 0;   // 1=VAI / 2=SIN VA / 3=Bestehorn VAJ
         Test : Struct
            ModeActive : Bool := false;   // mode test active (move between testpos 1 and 2)
            TarPos : Real := 5.0;   // target positon [mm]
            TarPos1 : Real := 5.0;   // target positon 1 [mm]
            TarPos2 : Real := 155.0;   // target positon 2 [mm]
            TimePosOk : Time := T#2s;   // time for position ok to switch to other position
         END_STRUCT;
         VAI : Struct
            Par1 : Real := 50.0;   // target positon [mm]
            Par2 : Real := 2.0;   // maximal velocity [m/s]
            Par3 : Real := 12.0;   // acceleration [m/s²]
            Par4 : Real := 12.0;   // deceleration [m/s²]
         END_STRUCT;
         SinVA : Struct
            Par1 : Real := 50.0;   // target positon [mm]
            Par2 : Real := 2.0;   // maximal velocity [m/s]
            Par3 : Real := 18.0;   // maixmal acceleration/deceleration [m/s²]
            Par4 : Real := 0.0;   // not used
         END_STRUCT;
         BestehornVAJ : Struct
            Par1 : Real := 50.0;   // target positon [mm]
            Par2 : Real := 2.0;   // maximal velocity [m/s]
            Par3 : Real := 24.0;   // maixmal acceleration/deceleration [m/s²]
            Par4 : Real := 450.0;   // maximal jerk [m/s³]
         END_STRUCT;
         Current : Struct   // current monitoring
            Man : Struct   // manual mode
               War : Struct
                  MinValue : Real := -3.0;   // min current value
                  MaxValue : Real := 2.0;   // max current value
                  Err : Bool;   // warning error
               END_STRUCT;
               Err : Struct
                  MinValue : Real := -3.0;   // min current value
                  MaxValue : Real := 2.0;   // max current value
                  Err : Bool;   // error
               END_STRUCT;
            END_STRUCT;
            Auto : Struct   // auto mode
               War : Struct
                  MinValue : Real := -15.0;   // min current value
                  MaxValue : Real := 16.0;   // max current value
                  Err : Bool;   // warning error
               END_STRUCT;
               Err : Struct
                  MinValue : Real := -15.0;   // min current value
                  MaxValue : Real := 16.0;   // max current value
                  Err : Bool;   // error
               END_STRUCT;
            END_STRUCT;
         END_STRUCT;
      END_STRUCT;
   END_VAR
BEGIN
END_DATA_BLOCK

DATA_BLOCK "Ref"   // DB600
{ S7_Optimized_Access := 'TRUE' }
// stored: AutoNumber false, IsRetainMemResEnabled true, MemoryReserve 500, RetainMemoryReserve 500
   VAR RETAIN
      adjTopCalOffset : DInt := -300;   // adjustment top calibration offset [mm/10]
      adjLeftCalOffset : DInt := 150;   // adjustment left calibration offset [mm/10]
      adjRightCalOffset : DInt := 101;   // adjustment right calibration offset [mm/10]
      adjScannerTar : Real := 60.0;   // adjustment scanner target position [mm/10]
      adjTopTar : Real := 12.0;   // adjustment top target position [mm/10]
      adjLeftTar : Real := 87.5;   // adjustment left target position [mm/10]
      adjRightTar : Real := 82.6;   // adjustment right target position [mm/10]
      adjScannerAct : DInt := -2135;   // adjustment scanner target position [mm/10]
      adjTopAct : DInt := -30;   // adjustment top target position [mm/10]
      adjLeftAct : DInt := 825;   // adjustment left target position [mm/10]
      adjRightAct : DInt := 825;   // adjustment right target position [mm/10]
      senTopCalOffset : Real := 0.0;   // sensor top calibration offset [mm]
      senLeftCalOffset : Real := 0.0;   // sensor left calibration offset [mm]
      senRightCalOffset : Real := 0.0;   // sensor right calibration offset [mm]
   END_VAR
BEGIN
END_DATA_BLOCK

ORGANIZATION_BLOCK "Main"   // OB1, FBD, ProgramCycle
TITLE = "Main Program Sweep (Cycle)"
{ S7_Optimized_Access := 'TRUE' }
// stored: SetENOAutomatically false
   VAR_INPUT
      Initial_Call : Bool;   // Initial call of this OB
      Remanence : Bool;   // =True, if remanent data are available
   END_VAR
   VAR_TEMP
      EV_CLASS : Byte;   // Bits 0-3 = 1:Coming event, Bits 4-7 = 1:Event class 1
      SCAN_1 : Byte;   // 1:Initial call of the OB, 3: Call 2-n of the OB
      PRIORITY : Byte;   // Priority of OB Execution
      OB_NUMBR : Byte;   // OB number
      RESERVED_1 : Byte;   // Reserved for system
      RESERVED_2 : Byte;   // Reserved for system
      PREV_CYCLE : Int;   // Previous program cycle time (milliseconds)
      MIN_CYCLE : Int;   // Minimum program cycle time (milliseconds)
      MAX_CYCLE : Int;   // Maximum program cycle time (milliseconds)
      DATE_TIME : Date_And_Time;   // Date and time OB started
      tempLreal : LReal;
   END_VAR
   VAR_TEMP   // added for the SCL form of the ladder/FBD networks
      _w1 : Bool;
      _s5time1 : S5Time;
      _w2 : Bool;
      _s5time2 : S5Time;
   END_VAR
BEGIN

NETWORK
TITLE = restart
      A     "firstScan";
      L     s5t#2s;
      SD    "T0";
      A     "T0";
      R     "firstScan";

NETWORK
TITLE = true/false test1/test0
      AN    "true";
      S     "true";
      A     "false";
      R     "false";

      AN    "test1";
      S     "test1";
      A     "test0";
      R     "test0";

      AN    "test1ibn";
      S     "test1ibn";
      A     "test0ibn";
      R     "test0ibn";


NETWORK
TITLE = clocks
      L     "systemClockByte";
      T     "clockByte";

      L     "cycleFlag";
      L     1;
      +I;
      T     "cycleFlag";

REGION Network 4: if you will test safety areas let run the plant in slow speed an set this tag
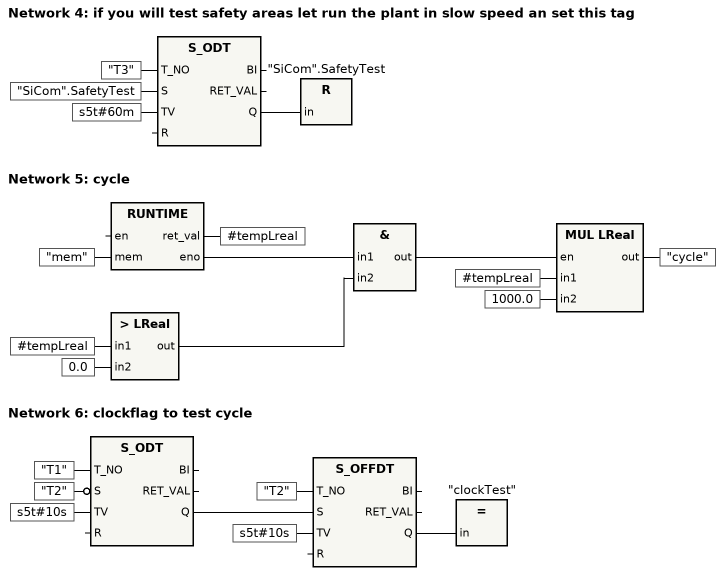
   #_s5time1 := S_ODT(T_NO := "T3", S := "SiCom".SafetyTest, TV := s5t#60m, Q => #_w1);
   IF #_w1 THEN "SiCom".SafetyTest := FALSE; END_IF;
END_REGION

REGION Network 5: cycle
   // no SCL statement known for Runtime: written as a call
   // ENO of a box is taken as its EN; it also drops when the box reports an error
   #tempLreal := Runtime(mem := "mem");
   IF #tempLreal > 0.0 THEN "cycle" := #tempLreal * 1000.0; END_IF;
END_REGION

REGION Network 6: clockflag to test cycle
   #_s5time1 := S_ODT(T_NO := "T1", S := NOT "T2", TV := s5t#10s, Q => #_w1);
   #_s5time2 := S_OFFDT(T_NO := "T2", S := #_w1, TV := s5t#10s, Q => #_w2);
   "clockTest" := #_w2;
END_REGION

NETWORK
TITLE = call instance

// Safety
      CALL  "SafetyCom", "SafetyCom_DB";

// Communication
      CALL  "Com", "Com_DB";

// General
      CALL  "Clock", "Clock_DB";
      CALL  "AutoIndication", "AutoIndication_DB";
      CALL  "Fault", "Fault_DB";
      CALL  "TestIo", "TestIo_DB";
      CALL  "ErrCom", "ErrCom_DB";

// Goldeneye
      CALL  "DataTakeOver", "DataTakeOver_DB";
      CALL  "Sensors", "Sensors_DB";
      CALL  "AdjScanner", "AdjScanner_DB";
      CALL  "AdjTop", "AdjTop_DB";
      CALL  "AdjLeft", "AdjLeft_DB";
      CALL  "AdjRight", "AdjRight_DB";
      CALL  "BlowOffValve", "BlowOffValve_DB";
      CALL  "AirConditioner", "AirConditioner_DB";

END_ORGANIZATION_BLOCK

FUNCTION_BLOCK "SafetyCom"   // FB45, FBD
{ S7_Optimized_Access := 'TRUE' }
// stored: AutoNumber false, MemoryReserve 100, SetENOAutomatically false
   VAR DB_SPECIFIC
      Var { ExternalAccessible := 'False'; ExternalVisible := 'False'; ExternalWritable := 'False'} : "TypeVar";
   END_VAR
BEGIN

REGION Network 1 (SCL): reset important data if communication is not working
   IF "G".errComPc THEN
       "ComRd".Data.safety.AreaAdjustmentOn := FALSE;
       "ComRd".Data.safety.AreaLaserOn := FALSE;
       "ComRd".Data.safety.AreaXrayOn  := FALSE;
       "ComRd".Data.safety.ResetSafetyDevice := FALSE;
   END_IF;
END_REGION

REGION Network 2 (SCL): safety program - copy data
   "SiCom".Ack := "G".ack;
   "SiCom".Blinker := "blinker";
   "SiCom".Flash := "flash";
   "SiCom".LampTest.SettingMode:= "ComRd".Data.TestOutput.Active AND "ComRd".Data.TestOutput."Q900.1";
   "SiCom".LampTest.LaserOn := "ComRd".Data.TestOutput.Active AND "ComRd".Data.TestOutput."Q908.0";
   "SiCom".LampTest.XrayOn := "ComRd".Data.TestOutput.Active AND "ComRd".Data.TestOutput."Q908.1";
   "SiCom".SafetyTest := false;

   "SiCom".AreaAdjustmentOn := "ComRd".Data.safety.AreaAdjustmentOn OR TRUE;
   "SiCom".AreaLaserOn := "ComRd".Data.safety.AreaLaserOn;
   "SiCom".AreaXrayOn := "ComRd".Data.safety.AreaXrayOn;

   "SiCom".ResetSafetyDevice := "ComRd".Data.safety.ResetSafetyDevice OR "G".ack;
END_REGION
END_FUNCTION_BLOCK

FUNCTION_BLOCK "Com"   // FB301, FBD
{ S7_Optimized_Access := 'FALSE' }
// stored: AutoNumber false, SetENOAutomatically false
   VAR
      Var { S7_SetPoint := 'True'} : "TypeVar";
      T : Array[1..6] of IEC_TIMER;
      wdOldParam { ExternalAccessible := 'False'; ExternalVisible := 'False'; ExternalWritable := 'False'} : Int;
      wdOldErr { ExternalAccessible := 'False'; ExternalVisible := 'False'; ExternalWritable := 'False'} : Int;
   END_VAR
   VAR_TEMP   // added for the SCL form of the ladder/FBD networks
      _w1 : Bool;
   END_VAR
BEGIN

REGION Network 1 (SCL): version info
   "ComSd".Data.config.Version := 13;

   IF "ComRd".Data.Config.version <> "ComSd".Data.config.Version THEN
       "G".errVersion := TRUE;
   ELSE
       "G".errVersion := FALSE;
   END_IF;

   IF "G".ack THEN
       "G".errVersion := FALSE;
   END_IF;
END_REGION

REGION Network 2: valid
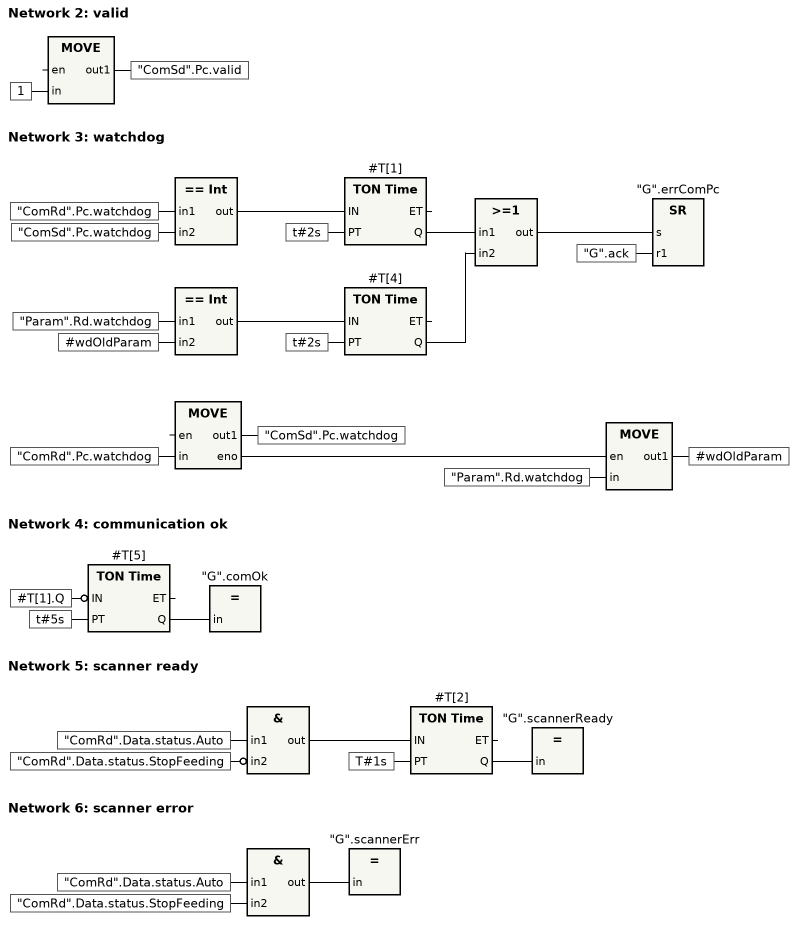
   "ComSd".Pc.valid := 1;
END_REGION

REGION Network 3: watchdog
   #T[1].TON(IN := "ComRd".Pc.watchdog = "ComSd".Pc.watchdog, PT := t#2s);
   #_w1 := #T[1].Q;
   #T[4].TON(IN := "Param".Rd.watchdog = #wdOldParam, PT := t#2s);
   IF #_w1 OR #T[4].Q THEN
       "G".errComPc := TRUE;   // SR flip-flop
   END_IF;
   IF "G".ack THEN "G".errComPc := FALSE; END_IF;
   "ComSd".Pc.watchdog := "ComRd".Pc.watchdog;
   #wdOldParam := "Param".Rd.watchdog;
END_REGION

REGION Network 4: communication ok
   #T[5].TON(IN := NOT #T[1].Q, PT := t#5s);
   "G".comOk := #T[5].Q;
END_REGION

REGION Network 5: scanner ready
   #T[2].TON(IN := "ComRd".Data.status.Auto AND NOT "ComRd".Data.status.StopFeeding, PT := T#1s);
   "G".scannerReady := #T[2].Q;
END_REGION

REGION Network 6: scanner error
   "G".scannerErr := "ComRd".Data.status.Auto AND "ComRd".Data.status.StopFeeding;
END_REGION

REGION Network 7: release infeed
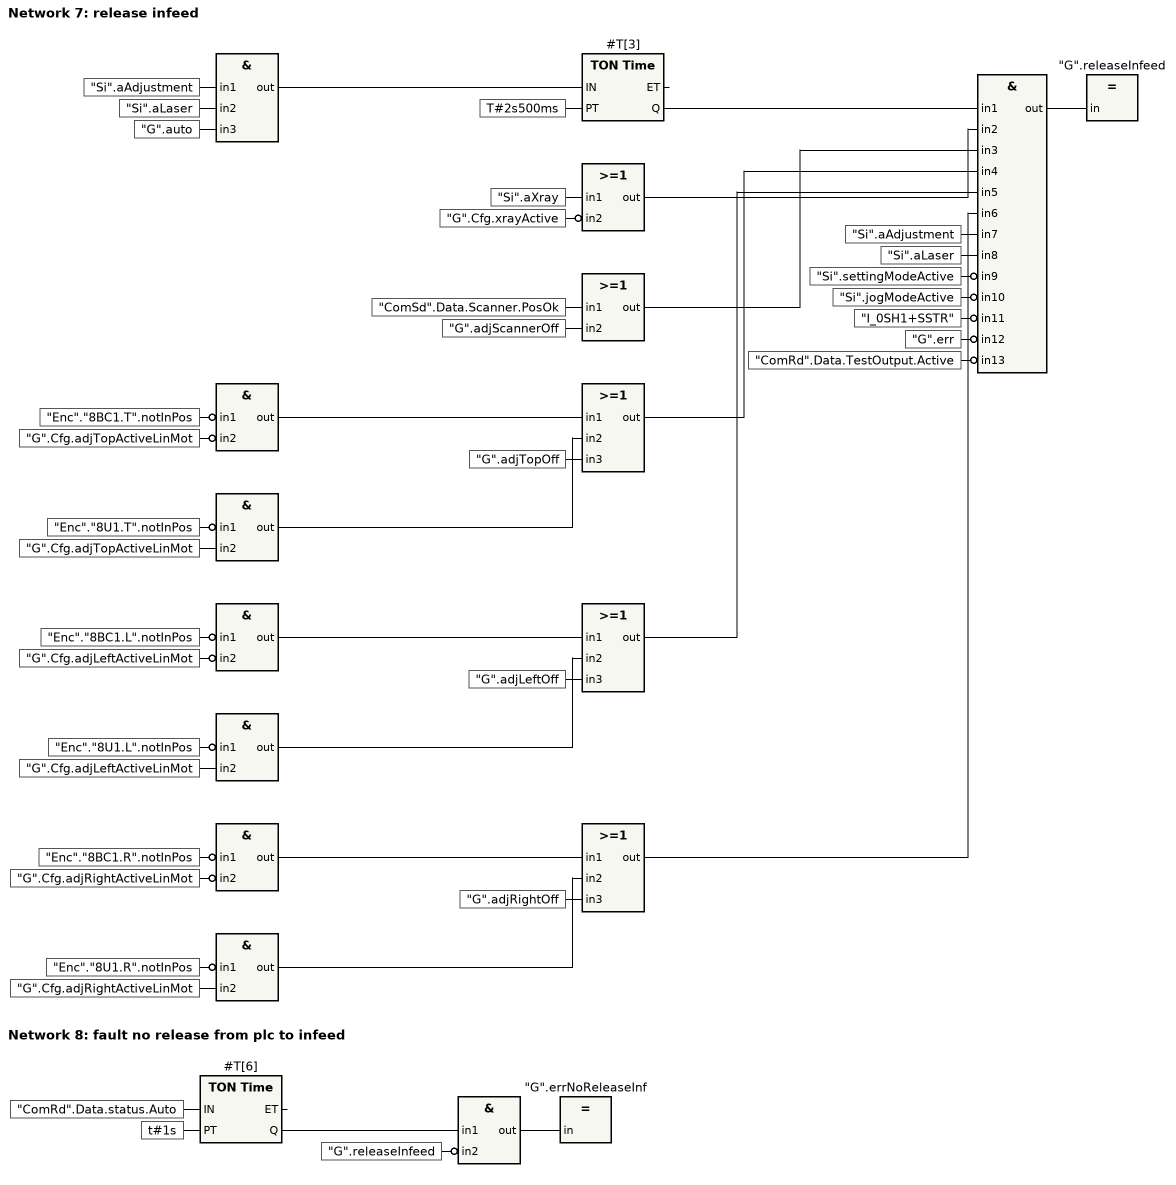
   #T[3].TON(IN := "Si".aAdjustment AND "Si".aLaser AND "G".auto, PT := T#2s500ms);
   "G".releaseInfeed := #T[3].Q AND ("Si".aXray OR NOT "G".Cfg.xrayActive) AND ("ComSd".Data.Scanner.PosOk OR "G".adjScannerOff) AND ((NOT "Enc"."8BC1.T".notInPos AND NOT "G".Cfg.adjTopActiveLinMot) OR (NOT "Enc"."8U1.T".notInPos AND "G".Cfg.adjTopActiveLinMot) OR "G".adjTopOff) AND ((NOT "Enc"."8BC1.L".notInPos AND NOT "G".Cfg.adjLeftActiveLinMot) OR (NOT "Enc"."8U1.L".notInPos AND "G".Cfg.adjLeftActiveLinMot) OR "G".adjLeftOff) AND ((NOT "Enc"."8BC1.R".notInPos AND NOT "G".Cfg.adjRightActiveLinMot) OR (NOT "Enc"."8U1.R".notInPos AND "G".Cfg.adjRightActiveLinMot) OR "G".adjRightOff) AND "Si".aAdjustment AND "Si".aLaser AND NOT "Si".settingModeActive AND NOT "Si".jogModeActive AND NOT "I_0SH1+SSTR" AND NOT "G".err AND NOT "ComRd".Data.TestOutput.Active;
END_REGION

REGION Network 8: fault no release from plc to infeed
   #T[6].TON(IN := "ComRd".Data.status.Auto, PT := t#1s);
   "G".errNoReleaseInf := #T[6].Q AND NOT "G".releaseInfeed;
END_REGION

REGION Network 9: communication signals
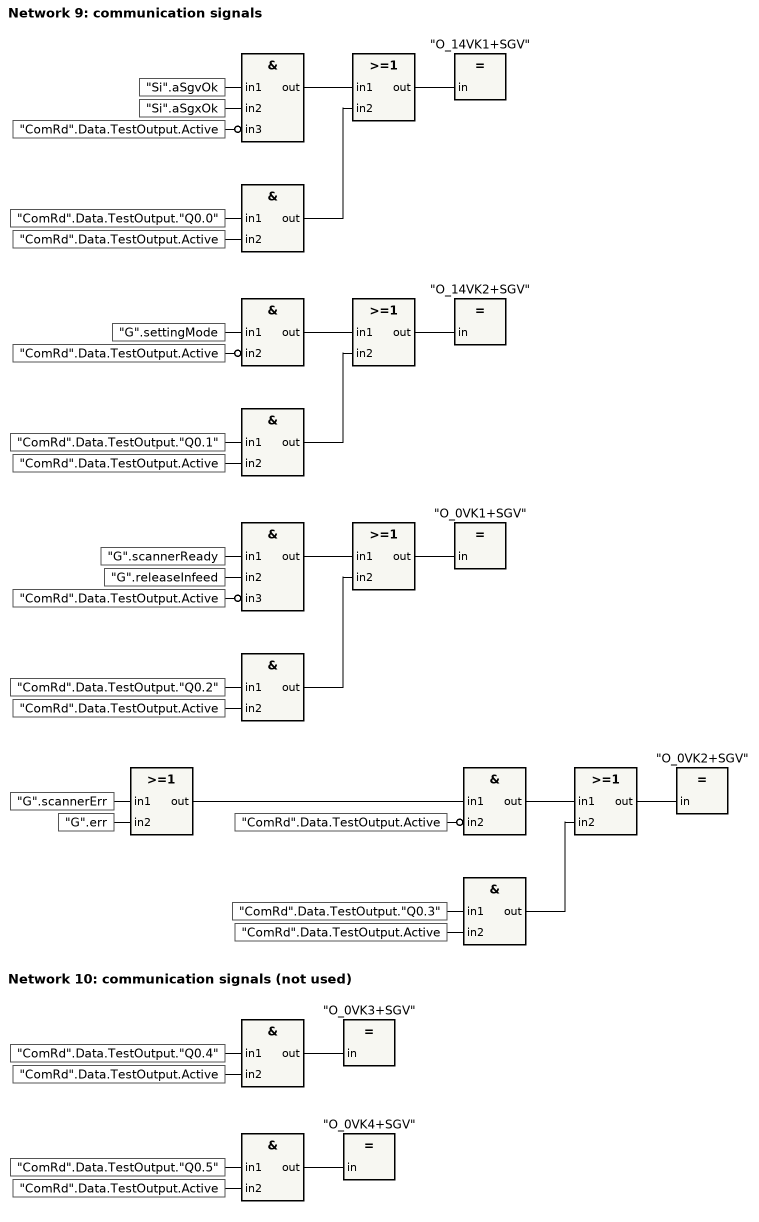
   "O_14VK1+SGV" := ("Si".aSgvOk AND "Si".aSgxOk AND NOT "ComRd".Data.TestOutput.Active) OR ("ComRd".Data.TestOutput."Q0.0" AND "ComRd".Data.TestOutput.Active);
   "O_14VK2+SGV" := ("G".settingMode AND NOT "ComRd".Data.TestOutput.Active) OR ("ComRd".Data.TestOutput."Q0.1" AND "ComRd".Data.TestOutput.Active);
   "O_0VK1+SGV" := ("G".scannerReady AND "G".releaseInfeed AND NOT "ComRd".Data.TestOutput.Active) OR ("ComRd".Data.TestOutput."Q0.2" AND "ComRd".Data.TestOutput.Active);
   "O_0VK2+SGV" := (("G".scannerErr OR "G".err) AND NOT "ComRd".Data.TestOutput.Active) OR ("ComRd".Data.TestOutput."Q0.3" AND "ComRd".Data.TestOutput.Active);
END_REGION

REGION Network 10: communication signals (not used)
   "O_0VK3+SGV" := "ComRd".Data.TestOutput."Q0.4" AND "ComRd".Data.TestOutput.Active;
   "O_0VK4+SGV" := "ComRd".Data.TestOutput."Q0.5" AND "ComRd".Data.TestOutput.Active;
END_REGION

REGION Network 11 (SCL): send
   // data - safety
   "ComSd".Data.safety.AreaAdjustmentOn := "Si".aAdjustment;
   "ComSd".Data.safety.AreaLaserOn := "Si".aLaser;
   "ComSd".Data.safety.AreaXrayOn := "Si".aXray;

   // data - status
   "ComSd".Data.status.err := "G".err;
   "ComSd".Data.status.ready := "G".scannerReady AND "G".releaseInfeed;
END_REGION
END_FUNCTION_BLOCK

FUNCTION_BLOCK "Clock"   // FB50, FBD
{ S7_Optimized_Access := 'FALSE' }
// stored: AutoNumber false, SetENOAutomatically false
   VAR
      Var { ExternalAccessible := 'False'; ExternalVisible := 'False'; ExternalWritable := 'False'} : "TypeVar";
      opHoRun { ExternalAccessible := 'False'; ExternalVisible := 'False'; ExternalWritable := 'False'} : Bool;
   END_VAR
   VAR_TEMP   // added for the SCL form of the ladder/FBD networks
      _w1 : Bool;
      _w2 : Bool;
   END_VAR
BEGIN

REGION Network 1: read date & time / Zeit lesen
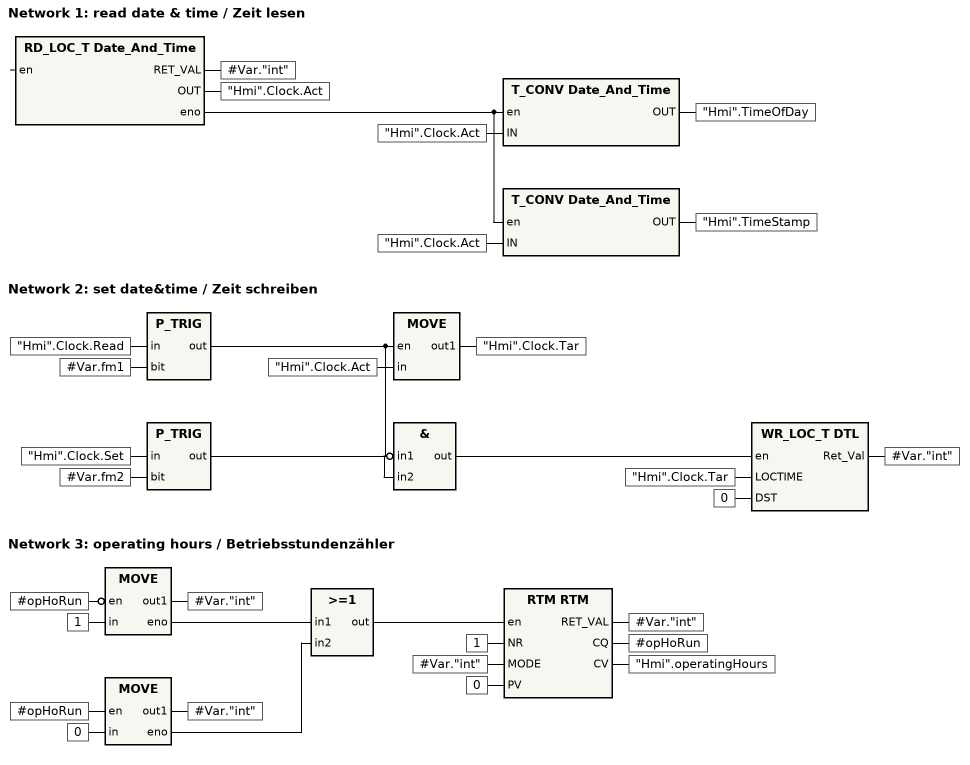
   #Var."int" := RD_LOC_T(OUT => "Hmi".Clock.Act, ENO => #_w1);
   IF #_w1 THEN
       T_CONV(IN := "Hmi".Clock.Act, OUT => "Hmi".TimeOfDay);
       T_CONV(IN := "Hmi".Clock.Act, OUT => "Hmi".TimeStamp);
   END_IF;
END_REGION

REGION Network 2: set date&time / Zeit schreiben
   #_w1 := "Hmi".Clock.Read AND NOT #Var.fm1;   // rising edge
   #Var.fm1 := "Hmi".Clock.Read;
   IF #_w1 THEN "Hmi".Clock.Tar := "Hmi".Clock.Act; END_IF;
   #_w2 := "Hmi".Clock.Set AND NOT #Var.fm2;   // rising edge
   #Var.fm2 := "Hmi".Clock.Set;
   IF NOT #_w1 AND #_w2 THEN #Var."int" := WR_LOC_T(LOCTIME := "Hmi".Clock.Tar, DST := 0); END_IF;
END_REGION

REGION Network 3: operating hours / Betriebsstundenzähler
   IF NOT #opHoRun THEN #Var."int" := 1; END_IF;
   IF #opHoRun THEN #Var."int" := 0; END_IF;
   IF NOT #opHoRun OR #opHoRun THEN
       #Var."int" := RTM(NR := 1, MODE := #Var."int", PV := 0, CQ => #opHoRun, CV => "Hmi".operatingHours);
   END_IF;
END_REGION
END_FUNCTION_BLOCK

FUNCTION_BLOCK "AutoIndication"   // FB300, FBD
{ S7_Optimized_Access := 'TRUE' }
// stored: AutoNumber false, MemoryReserve 100, SetENOAutomatically false
   VAR DB_SPECIFIC
      Var { ExternalAccessible := 'False'; ExternalVisible := 'False'; ExternalWritable := 'False'} : "TypeVar";
      T { ExternalAccessible := 'False'; ExternalVisible := 'False'; ExternalWritable := 'False'} : Array[1..5] of IEC_TIMER;
   END_VAR
BEGIN

REGION Network 1: lamp test
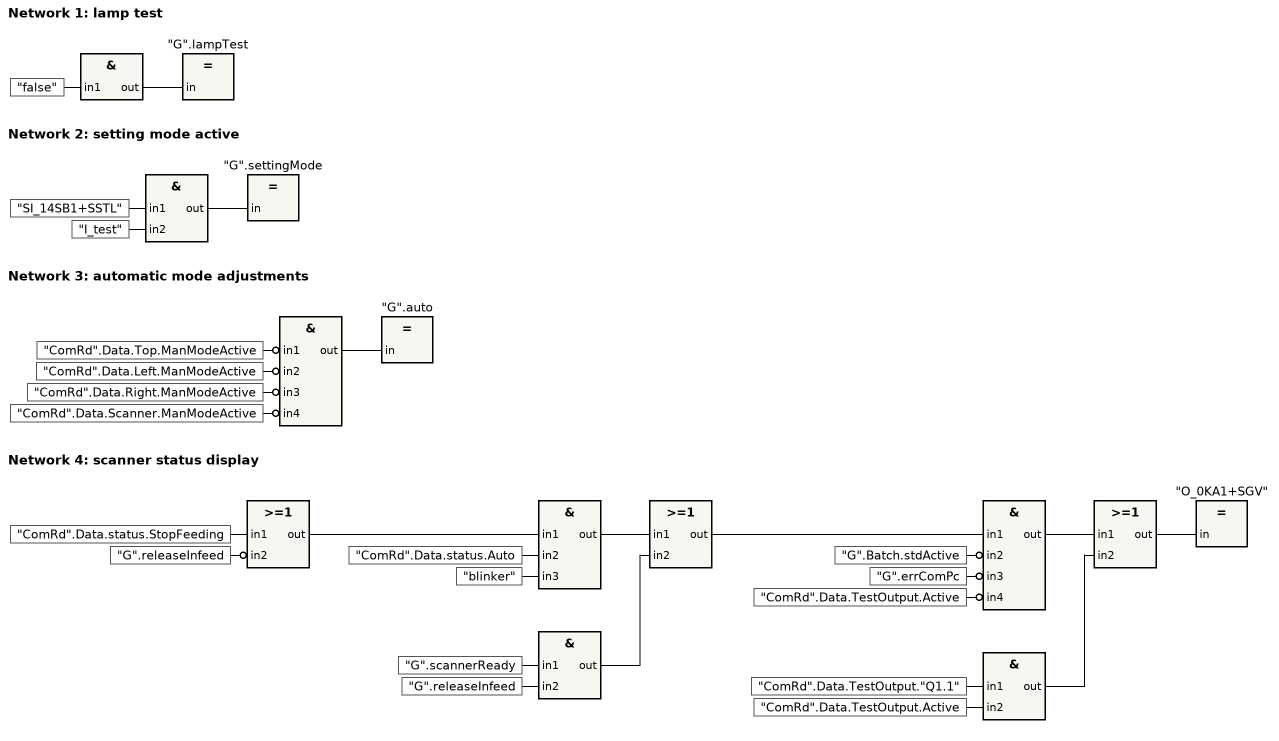
   "G".lampTest := "false";
END_REGION

REGION Network 2: setting mode active
   "G".settingMode := "SI_14SB1+SSTL" AND "I_test";
END_REGION

REGION Network 3: automatic mode adjustments
   "G".auto := NOT "ComRd".Data.Top.ManModeActive AND NOT "ComRd".Data.Left.ManModeActive AND NOT "ComRd".Data.Right.ManModeActive AND NOT "ComRd".Data.Scanner.ManModeActive;
END_REGION

REGION Network 4: scanner status display
   "O_0KA1+SGV" := (((("ComRd".Data.status.StopFeeding OR NOT "G".releaseInfeed) AND "ComRd".Data.status.Auto AND "blinker") OR ("G".scannerReady AND "G".releaseInfeed)) AND NOT "G".Batch.stdActive AND NOT "G".errComPc AND NOT "ComRd".Data.TestOutput.Active) OR ("ComRd".Data.TestOutput."Q1.1" AND "ComRd".Data.TestOutput.Active);
END_REGION
END_FUNCTION_BLOCK

FUNCTION_BLOCK "Fault"   // FB304, FBD
{ S7_Optimized_Access := 'TRUE' }
// stored: AutoNumber false, MemoryReserve 100, SetENOAutomatically false
   VAR
      Var : "TypeVar";
      T : Array[1..16] of IEC_TIMER;
      ErrSafetyModule { ExternalAccessible := 'False'; ExternalVisible := 'False'; ExternalWritable := 'False'} : Bool;
   END_VAR
BEGIN

REGION Network 1: fault acknowledge - pc
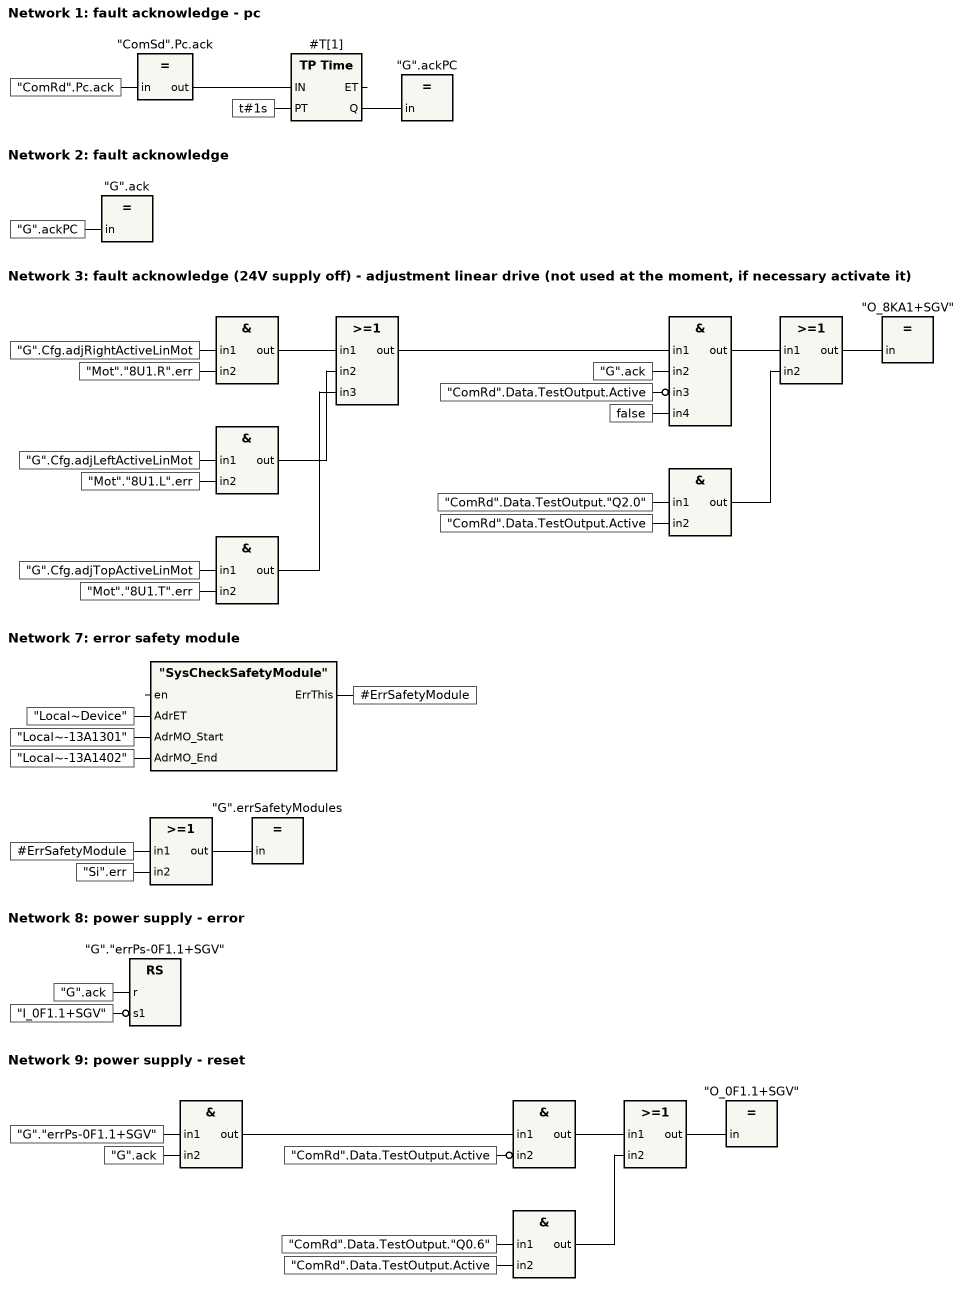
   "ComSd".Pc.ack := "ComRd".Pc.ack;
   #T[1].TP(IN := "ComRd".Pc.ack, PT := t#1s);
   "G".ackPC := #T[1].Q;
END_REGION

REGION Network 2: fault acknowledge
   "G".ack := "G".ackPC;
END_REGION

REGION Network 3: fault acknowledge (24V supply off) - adjustment linear drive (not used at the moment, if necessary activate it)
   "O_8KA1+SGV" := ((("G".Cfg.adjRightActiveLinMot AND "Mot"."8U1.R".err) OR ("G".Cfg.adjLeftActiveLinMot AND "Mot"."8U1.L".err) OR ("G".Cfg.adjTopActiveLinMot AND "Mot"."8U1.T".err)) AND "G".ack AND NOT "ComRd".Data.TestOutput.Active AND false) OR ("ComRd".Data.TestOutput."Q2.0" AND "ComRd".Data.TestOutput.Active);
END_REGION

NETWORK
TITLE = info general
      O     "false";

      =     "G".info;

NETWORK
TITLE = warning general
      O     "Si".settingModeActive;
      O     "Si".jogModeActive;
      O     "I_0SH1+SSTR";

      =     "G".war;

NETWORK
TITLE = fault general
// fault safety
      O     "G".errSafetyModules;
      O     "Si".aLaserErrFdb;
      O     "Si".aAdjustmentErrFdb1;
      O     "Si".aAdjustmentErrFdb2;
      O(;
      A     "Si".aXrayErrFdb;
      A     "G".Cfg.xrayActive;
      );

// fault communication / pc
      O     "G".errComPc;
      O     "G".errVersion;

// fault power supply
      O     "G"."errPs-0F1.1+SGV";
      O     "G"."errAc-0E1+SGV";
      O     "G"."errAc-0E2+SGX";
      O     "G"."errAc-0E1.1+SGV";

// fault profinet
      O     "G".errProfinet;

// fault sensor
      O     "Sen"."1BTR2+SGV".err;
      O     "Sen"."1BTR2+SGX".err;

// fault encoder
      O     "Enc"."1BCI1".err;
      O     "Enc"."1BCM1".err;
      O     "Enc"."1BCO1".err;

// fault motor
      O     "G".errAdjScanner;
      O     "G".errAdjTop;
      O     "G".errAdjLeft;
      O     "G".errAdjRight;

      O     "false";
      =     "G".err;

REGION Network 7: error safety module
   "SysCheckSafetyModule"(AdrET := "Local~Device",
                          AdrMO_Start := "Local~-13A1301",
                          AdrMO_End := "Local~-13A1402",
                          ErrThis => #ErrSafetyModule);
   "G".errSafetyModules := #ErrSafetyModule OR "Si".err;
END_REGION

REGION Network 8: power supply - error
   IF "G".ack THEN
       "G"."errPs-0F1.1+SGV" := FALSE;   // RS flip-flop
   END_IF;
   IF NOT "I_0F1.1+SGV" THEN "G"."errPs-0F1.1+SGV" := TRUE; END_IF;
END_REGION

REGION Network 9: power supply - reset
   "O_0F1.1+SGV" := ("G"."errPs-0F1.1+SGV" AND "G".ack AND NOT "ComRd".Data.TestOutput.Active) OR ("ComRd".Data.TestOutput."Q0.6" AND "ComRd".Data.TestOutput.Active);
END_REGION

REGION Network 10: fault profinet device
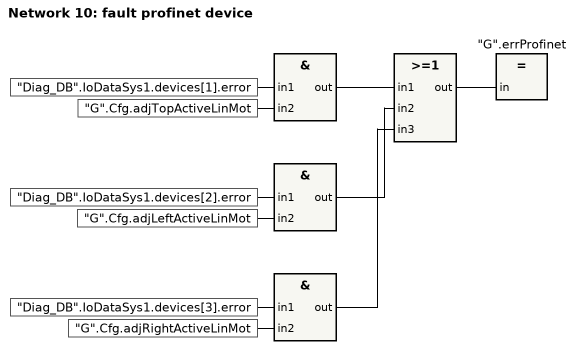
   "G".errProfinet := ("Diag_DB".IoDataSys1.devices[1].error AND "G".Cfg.adjTopActiveLinMot) OR ("Diag_DB".IoDataSys1.devices[2].error AND "G".Cfg.adjLeftActiveLinMot) OR ("Diag_DB".IoDataSys1.devices[3].error AND "G".Cfg.adjRightActiveLinMot);
END_REGION
END_FUNCTION_BLOCK

FUNCTION "SysCheckSafetyModule" : Void   // FC2157, FBD
TITLE = SysCheckSafetyModules
{ S7_Optimized_Access := 'TRUE' }
// stored: AutoNumber false, SetENOAutomatically false
   VAR_INPUT
      AdrET : HW_DEVICE;   // Address of the ET station
      AdrMO_Start : HW_IO;   // Address of first ET modul
      AdrMO_End : HW_IO;   // Address of last ET modul
   END_VAR
   VAR_OUTPUT
      ErrThis : Bool;
   END_VAR
   VAR_TEMP
      i : Int;
      tFirstSlot : Int;
      tLastSlot : Int;
      t_Err : Bool;
      t_RetVal : Int;
      tState : Array[0..127] of Bool;
      tGeoAddr : GEOADDR;
   END_VAR
   VAR_TEMP   // added for the SCL form of the ladder/FBD networks
      _w1 : Bool;
      _w2 : Bool;
   END_VAR
BEGIN

REGION Network 1: read module slot numbers
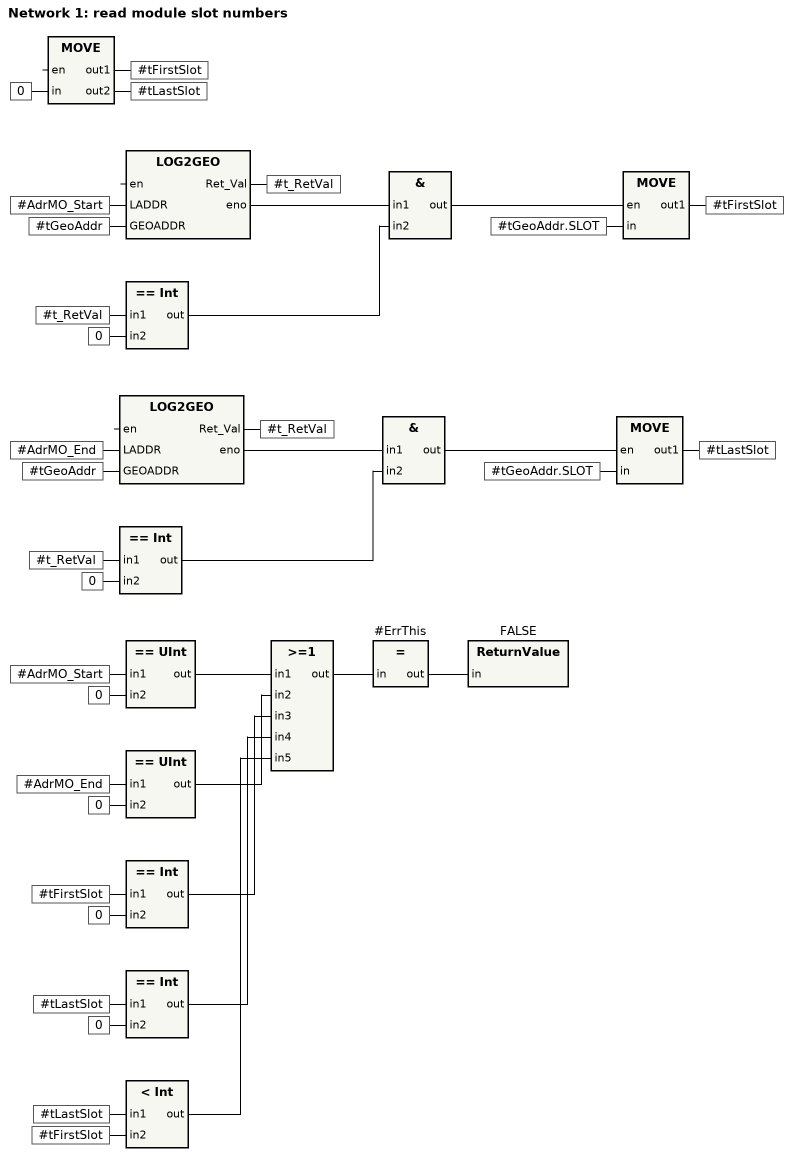
   #tFirstSlot := 0;
   #tLastSlot := 0;
   #t_RetVal := LOG2GEO(LADDR := #AdrMO_Start, GEOADDR := #tGeoAddr, ENO => #_w1);
   IF #_w1 AND (#t_RetVal = 0) THEN #tFirstSlot := #tGeoAddr.SLOT; END_IF;
   #t_RetVal := LOG2GEO(LADDR := #AdrMO_End, GEOADDR := #tGeoAddr, ENO => #_w2);
   IF #_w2 AND (#t_RetVal = 0) THEN #tLastSlot := #tGeoAddr.SLOT; END_IF;
   #ErrThis := (#AdrMO_Start = 0) OR (#AdrMO_End = 0) OR (#tFirstSlot = 0) OR (#tLastSlot = 0) OR (#tLastSlot < #tFirstSlot);
   IF #ErrThis THEN
       ENO := FALSE;
       RETURN;
   END_IF;
END_REGION

REGION Network 2: read station status
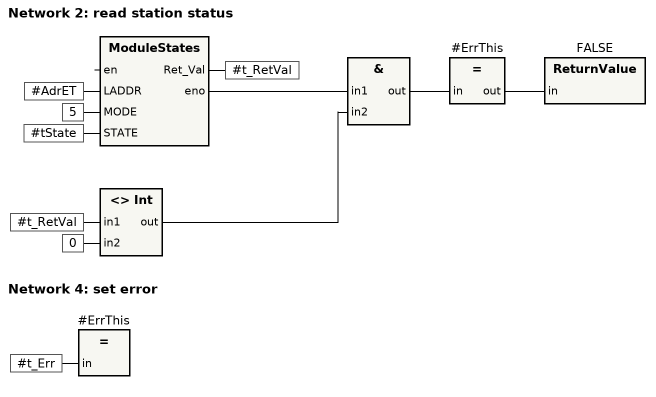
   #t_RetVal := ModuleStates(LADDR := #AdrET, MODE := 5, STATE := #tState, ENO => #_w1);
   #ErrThis := #_w1 AND (#t_RetVal <> 0);
   IF #ErrThis THEN
       ENO := FALSE;
       RETURN;
   END_IF;
END_REGION

REGION Network 3 (SCL): search for fault
   #t_Err := false;
   FOR #i := #tFirstSlot TO #tLastSlot DO
       IF #tState[#i+1] THEN
           #t_Err := true;
           EXIT;
       END_IF;
   END_FOR;
END_REGION

REGION Network 4: set error
   #ErrThis := #t_Err;
END_REGION
END_FUNCTION

FUNCTION_BLOCK "TestIo"   // FB306, FBD
{ S7_Optimized_Access := 'TRUE' }
// stored: AutoNumber false, MemoryReserve 100, SetENOAutomatically false
BEGIN

REGION Network 1 (SCL): Data PLC Input Normal

   "ComSd".Data.PlcInputNormal."I0.0" := "I_IN1_EXT+SGV";
   "ComSd".Data.PlcInputNormal."I0.1" := "I_IN2_EXT+SGV";
   "ComSd".Data.PlcInputNormal."I0.2" := "I_IN3_EXT+SGV";
   "ComSd".Data.PlcInputNormal."I0.3" := "I_0E1+SGV";
   "ComSd".Data.PlcInputNormal."I0.4" := "I_0E2+SGX";
   "ComSd".Data.PlcInputNormal."I0.5" := "I_0F1.1+SGV";
   "ComSd".Data.PlcInputNormal."I0.6" := "I_0SH1+SSTR";
   "ComSd".Data.PlcInputNormal."I0.7" := "I_14SB0+HMI";
   "ComSd".Data.PlcInputNormal."I1.0" := "I_14SB1+HMI";
   "ComSd".Data.PlcInputNormal."I1.1" := "I_8S1.T_in";
   "ComSd".Data.PlcInputNormal."I1.2" := "I_8S2.T_out";
   "ComSd".Data.PlcInputNormal."I1.3" := "I_8S1.L_in";
   "ComSd".Data.PlcInputNormal."I1.4" := "I_8S2.L_out";
   "ComSd".Data.PlcInputNormal."I1.5" := "I_8S1.R_in";
   "ComSd".Data.PlcInputNormal."I1.6" := "I_8S2.R_out";
   "ComSd".Data.PlcInputNormal."I1.7" := "I_1BTR2+SGV";
   "ComSd".Data.PlcInputNormal."I2.0" := "I_8S1.B_left";
   "ComSd".Data.PlcInputNormal."I2.1" := "I_8S2.B_right";
   "ComSd".Data.PlcInputNormal."I2.2" := "I_1BTR2+SGX";
   "ComSd".Data.PlcInputNormal."I2.3" := "I_0E1.1+SGV";
   "ComSd".Data.PlcInputNormal."I2.4" := "I_spare24";
   "ComSd".Data.PlcInputNormal."I2.5" := "I_spare25";
   "ComSd".Data.PlcInputNormal."I2.6" := "I_spare26";
   "ComSd".Data.PlcInputNormal."I2.7" := "I_spare27";
END_REGION

REGION Network 2 (SCL): Data PLC Input Safety

   "ComSd".Data.PlcInputSafety."I800.0" := "SI_NA_EXT+SGV";
   "ComSd".Data.PlcInputSafety."I800.1" := "SI_14SB0/1+HMI";
   "ComSd".Data.PlcInputSafety."I800.2" := "SI_14SB1+SSTL";
   "ComSd".Data.PlcInputSafety."I800.3" := "SI_14SB2+SSTL";
   "ComSd".Data.PlcInputSafety."I808.0" := "SI_14SS1.TL+SGV";
   "ComSd".Data.PlcInputSafety."I808.1" := "SI_14SS1.BL+SGV";
   "ComSd".Data.PlcInputSafety."I808.2" := "SI_14SS1.TR+SGV";
   "ComSd".Data.PlcInputSafety."I808.3" := "SI_14SS1.BR+SGV";
   "ComSd".Data.PlcInputSafety."I816.0" := "SI_14SS1.TL+SGX";
   "ComSd".Data.PlcInputSafety."I816.1" := "SI_14SS1.BL+SGX";
   "ComSd".Data.PlcInputSafety."I816.2" := "SI_14SS1.TR+SGX";
   "ComSd".Data.PlcInputSafety."I816.3" := "SI_14SS1.BR+SGX";
   "ComSd".Data.PlcInputSafety."I824.0" := "SI_8U1+SGV";
   "ComSd".Data.PlcInputSafety."I824.1" := "SI_14KA1+SGV";
   "ComSd".Data.PlcInputSafety."I824.2" := "SI_14KA2+SGV";
   "ComSd".Data.PlcInputSafety."I824.3" := "SI_5AX1+SGX";
END_REGION

REGION Network 3 (SCL): Data PLC Output Normal

